LIN {X 0,Y 181.096,Z 303.588,A -85,B 0,C 180,E1 -24675.57,E2 -24675.57} C_VEL
LIN {X 0,Y 183.725,Z 307.761,A -85,B 0,C 180,E1 -24677.82,E2 -24677.82} C_VEL
LIN {X 0,Y 187.642,Z 314.233,A -85,B 0,C 180,E1 -24680.781,E2 -24680.781} C_VEL
LIN {X 0,Y 192.444,Z 323.016,A -85,B 0,C 180,E1 -24683.954,E2 -24683.954} C_VEL
LIN {X 0,Y 193.88,Z 325.932,A -85,B 0,C 180,E1 -24684.834,E2 -24684.834} C_VEL
LIN {X 0,Y 191.762,Z 350.553,A -85,B 0,C 180,E1 -24685.67,E2 -24685.67} C_VEL
LIN {X 0,Y 189.631,Z 363.427,A -85,B 0,C 180,E1 -24686.415,E2 -24686.415} C_VEL
LIN {X 0,Y 186.579,Z 375.788,A -85,B 0,C 180,E1 -24687.439,E2 -24687.439} C_VEL
LIN {X 0,Y 182.556,Z 388.05,A -85,B 0,C 180,E1 -24688.863,E2 -24688.863} C_VEL
LIN {X 0,Y 178.131,Z 398.759,A -85,B 0,C 180,E1 -24690.531,E2 -24690.531} C_VEL
LIN {X 0,Y 173.052,Z 408.926,A -85,B 0,C 180,E1 -24692.579,E2 -24692.579} C_VEL
LIN {X 0,Y 167.41,Z 418.371,A -85,B 0,C 180,E1 -24695.058,E2 -24695.058} C_VEL
LIN {X 0,Y 161.166,Z 427.427,A -85,B 0,C 180,E1 -24698.291,E2 -24698.291} C_VEL
LIN {X 0,Y 155.369,Z 434.616,A -85,B 0,C 180,E1 -24701.728,E2 -24701.728} C_VEL
LIN {X 0,Y 150.26,Z 440.26,A -85,B 0,C 180,E1 -24705.45,E2 -24705.45} C_VEL
LIN {X 0,Y 145.741,Z 444.612,A -85,B 0,C 180,E1 -24709.387,E2 -24709.387} C_VEL
LIN {X 0,Y 141.866,Z 447.811,A -85,B 0,C 180,E1 -24713.529,E2 -24713.529} C_VEL
LIN {X 0,Y 139.709,Z 449.369,A -85,B 0,C 180,E1 -24716.407,E2 -24716.407} C_VEL
LIN {X 0,Y 137.256,Z 450.755,A -85,B 0,C 180,E1 -24720.514,E2 -24720.514} C_VEL
LIN {X 0,Y 135.153,Z 451.346,A -85,B 0,C 180,E1 -24725.421,E2 -24725.421} C_VEL
LIN {X 0,Y 133.809,Z 450.698,A -85,B 0,C 180,E1 -24730.983,E2 -24730.983} C_VEL
LIN {X 0,Y 133.388,Z 449.493,A -85,B 0,C 180,E1 -24734.729,E2 -24734.729} C_VEL
LIN {X 0,Y 133.321,Z 448.048,A -85,B 0,C 180,E1 -24737.831,E2 -24737.831} C_VEL
LIN {X 0,Y 133.812,Z 445.016,A -85,B 0,C 180,E1 -24742.458,E2 -24742.458} C_VEL
LIN {X 0,Y 134.775,Z 440.923,A -85,B 0,C 180,E1 -24747.014,E2 -24747.014} C_VEL
LIN {X 0,Y 136.471,Z 434.662,A -85,B 0,C 180,E1 -24752.217,E2 -24752.217} C_VEL
LIN {X 0,Y 138.593,Z 427.846,A -85,B 0,C 180,E1 -24756.555,E2 -24756.555} C_VEL
LIN {X 0,Y 141.366,Z 419.285,A -85,B 0,C 180,E1 -24760.748,E2 -24760.748} C_VEL
LIN {X 0,Y 144.499,Z 409.445,A -85,B 0,C 180,E1 -24764.473,E2 -24764.473} C_VEL
LIN {X 0,Y 147.424,Z 399.807,A -85,B 0,C 180,E1 -24767.293,E2 -24767.293} C_VEL
LIN {X 0,Y 150.331,Z 388.712,A -85,B 0,C 180,E1 -24769.815,E2 -24769.815} C_VEL
LIN {X 0,Y 152.82,Z 376.588,A -85,B 0,C 180,E1 -24771.944,E2 -24771.944} C_VEL
LIN {X 0,Y 154.786,Z 365,A -85,B 0,C 180,E1 -24773.412,E2 -24773.412} C_VEL
LIN {X 0,Y 156.38,Z 351.822,A -85,B 0,C 180,E1 -24774.555,E2 -24774.555} C_VEL
LIN {X 0,Y 157.472,Z 336.902,A -85,B 0,C 180,E1 -24775.295,E2 -24775.295} C_VEL
LIN {X 0,Y 159.848,Z 295.992,A -85,B 0,C 180,E1 -24776.933,E2 -24776.933} C_VEL
LIN {X 0,Y 157.515,Z 290.307,A -85,B 0,C 180,E1 -24777.849,E2 -24777.849} C_VEL
LIN {X 0,Y 151.057,Z 277.224,A -85,B 0,C 180,E1 -24780.433,E2 -24780.433} C_VEL
LIN {X 0,Y 143.732,Z 264.819,A -85,B 0,C 180,E1 -24783.62,E2 -24783.62} C_VEL
LIN {X 0,Y 141.087,Z 260.921,A -85,B 0,C 180,E1 -24784.855,E2 -24784.855} C_VEL
LIN {X 0,Y 138.626,Z 257.169,A -85,B 0,C 180,E1 -24786.079,E2 -24786.079} C_VEL
LIN {X 0,Y 136.758,Z 254.919,A -85,B 0,C 180,E1 -24787.006,E2 -24787.006} C_VEL
LIN {X 0,Y 136.034,Z 252.53,A -85,B 0,C 180,E1 -24787.53,E2 -24787.53} C_VEL
LIN {X 0,Y 135.984,Z 252.525,A -85,B 0,C 180,E1 -24793.65,E2 -24793.65} C_VEL
LIN {X 0,Y 135.989,Z 252.541,A -85,B 0,C 180,E1 -24797.789,E2 -24797.789} C_VEL
LIN {X 0,Y 136.026,Z 252.509,A -85,B 0,C 180,E1 -24801.683,E2 -24801.683} C_VEL
LIN {X 0,Y 136.061,Z 252.533,A -85,B 0,C 180,E1 -24805.741,E2 -24805.741} C_VEL
LIN {X 0,Y 136.344,Z 252.463,A -85,B 0,C 180,E1 -24810.946,E2 -24810.946} C_VEL
LIN {X 0,Y 139.989,Z 268.771,A -85,B 0,C 180,E1 -24812.601,E2 -24812.601} C_VEL
LIN {X 0,Y 142.664,Z 279.155,A -85,B 0,C 180,E1 -24813.601,E2 -24813.601} C_VEL
LIN {X 0,Y 139.563,Z 347.819,A -85,B 0,C 180,E1 -24820.511,E2 -24820.511} C_VEL
LIN {X 0,Y 138.874,Z 361.236,A -85,B 0,C 180,E1 -24822.323,E2 -24822.323} C_VEL
LIN {X 0,Y 137.939,Z 375.222,A -85,B 0,C 180,E1 -24824.863,E2 -24824.863} C_VEL
LIN {X 0,Y 137.171,Z 388.146,A -85,B 0,C 180,E1 -24827.906,E2 -24827.906} C_VEL
LIN {X 0,Y 136.431,Z 400.193,A -85,B 0,C 180,E1 -24831.482,E2 -24831.482} C_VEL
LIN {X 0,Y 136.056,Z 409.375,A -85,B 0,C 180,E1 -24834.813,E2 -24834.813} C_VEL
LIN {X 0,Y 135.846,Z 419.39,A -85,B 0,C 180,E1 -24839.258,E2 -24839.258} C_VEL
LIN {X 0,Y 135.797,Z 427.45,A -85,B 0,C 180,E1 -24843.709,E2 -24843.709} C_VEL
LIN {X 0,Y 136.499,Z 435.149,A -85,B 0,C 180,E1 -24848.885,E2 -24848.885} C_VEL
LIN {X 0,Y 137.925,Z 441.004,A -85,B 0,C 180,E1 -24853.702,E2 -24853.702} C_VEL
LIN {X 0,Y 140.845,Z 446.332,A -85,B 0,C 180,E1 -24858.925,E2 -24858.925} C_VEL
LIN {X 0,Y 144.451,Z 449.823,A -85,B 0,C 180,E1 -24862.906,E2 -24862.906} C_VEL
LIN {X 0,Y 150.485,Z 453.338,A -85,B 0,C 180,E1 -24867.841,E2 -24867.841} C_VEL
LIN {X 0,Y 157.818,Z 455.582,A -85,B 0,C 180,E1 -24872.302,E2 -24872.302} C_VEL
LIN {X 0,Y 166.371,Z 456.6,A -85,B 0,C 180,E1 -24876.256,E2 -24876.256} C_VEL
LIN {X 0,Y 175.918,Z 456.39,A -85,B 0,C 180,E1 -24879.732,E2 -24879.732} C_VEL
LIN {X 0,Y 186.402,Z 454.92,A -85,B 0,C 180,E1 -24882.739,E2 -24882.739} C_VEL
LIN {X 0,Y 184.858,Z 455.476,A -85,B 0,C 180,E1 -24883.748,E2 -24883.748} C_VEL
LIN {X 0,Y 174.305,Z 457.921,A -85,B 0,C 180,E1 -24886.726,E2 -24886.726} C_VEL
LIN {X 0,Y 164.675,Z 459.211,A -85,B 0,C 180,E1 -24890.192,E2 -24890.192} C_VEL
LIN {X 0,Y 156.122,Z 459.381,A -85,B 0,C 180,E1 -24894.179,E2 -24894.179} C_VEL
LIN {X 0,Y 149.087,Z 458.493,A -85,B 0,C 180,E1 -24898.762,E2 -24898.762} C_VEL
LIN {X 0,Y 143.43,Z 456.512,A -85,B 0,C 180,E1 -24903.829,E2 -24903.829} C_VEL
LIN {X 0,Y 139.429,Z 453.415,A -85,B 0,C 180,E1 -24909.336,E2 -24909.336} C_VEL
LIN {X 0,Y 137.239,Z 448.837,A -85,B 0,C 180,E1 -24915.635,E2 -24915.635} C_VEL
LIN {X 0,Y 135.307,Z 453.281,A -85,B 0,C 180,E1 -24919.522,E2 -24919.522} C_VEL
LIN {X 0,Y 134.113,Z 457.635,A -85,B 0,C 180,E1 -24924.66,E2 -24924.66} C_VEL
LIN {X 0,Y 134.086,Z 460.72,A -85,B 0,C 180,E1 -24929.997,E2 -24929.997} C_VEL
LIN {X 0,Y 133.697,Z 462.053,A -85,B 0,C 180,E1 -24933.976,E2 -24933.976} C_VEL
LIN {X 0,Y 132.967,Z 462.531,A -85,B 0,C 180,E1 -24936.491,E2 -24936.491} C_VEL
LIN {X 0,Y 130.508,Z 462.645,A -85,B 0,C 180,E1 -24940.674,E2 -24940.674} C_VEL
LIN {X 0,Y 128.888,Z 462.263,A -85,B 0,C 180,E1 -24944.118,E2 -24944.118} C_VEL
LIN {X 0,Y 128.744,Z 461.738,A -85,B 0,C 180,E1 -24946.746,E2 -24946.746} C_VEL
LIN {X 0,Y 129.013,Z 461.468,A -85,B 0,C 180,E1 -24947.611,E2 -24947.611} C_VEL
LIN {X 0,Y 131.421,Z 459.832,A -85,B 0,C 180,E1 -24951.98,E2 -24951.98} C_VEL
LIN {X 0,Y 134.738,Z 457.195,A -85,B 0,C 180,E1 -24956.315,E2 -24956.315} C_VEL
LIN {X 0,Y 139.233,Z 453.074,A -85,B 0,C 180,E1 -24960.897,E2 -24960.897} C_VEL
LIN {X 0,Y 145.186,Z 447.039,A -85,B 0,C 180,E1 -24965.509,E2 -24965.509} C_VEL
LIN {X 0,Y 150.9,Z 440.622,A -85,B 0,C 180,E1 -24968.954,E2 -24968.954} C_VEL
LIN {X 0,Y 157.14,Z 432.662,A -85,B 0,C 180,E1 -24972.13,E2 -24972.13} C_VEL
LIN {X 0,Y 162.721,Z 424.557,A -85,B 0,C 180,E1 -24974.571,E2 -24974.571} C_VEL
LIN {X 0,Y 168.557,Z 414.679,A -85,B 0,C 180,E1 -24976.854,E2 -24976.854} C_VEL
LIN {X 0,Y 173.526,Z 404.9,A -85,B 0,C 180,E1 -24978.523,E2 -24978.523} C_VEL
LIN {X 0,Y 178.054,Z 394.302,A -85,B 0,C 180,E1 -24979.881,E2 -24979.881} C_VEL
LIN {X 0,Y 182.319,Z 381.64,A -85,B 0,C 180,E1 -24981.085,E2 -24981.085} C_VEL
LIN {X 0,Y 185.37,Z 369.086,A -85,B 0,C 180,E1 -24981.926,E2 -24981.926} C_VEL
LIN {X 0,Y 187.487,Z 355.083,A -85,B 0,C 180,E1 -24982.545,E2 -24982.545} C_VEL
LIN {X 0,Y 189.689,Z 328.895,A -85,B 0,C 180,E1 -24983.386,E2 -24983.386} C_VEL
LIN {X 0,Y 185.015,Z 319.976,A -85,B 0,C 180,E1 -24986.684,E2 -24986.684} C_VEL
LIN {X 0,Y 180.62,Z 312.326,A -85,B 0,C 180,E1 -24990.306,E2 -24990.306} C_VEL
LIN {X 0,Y 177.664,Z 307.74,A -85,B 0,C 180,E1 -24993.13,E2 -24993.13} C_VEL
LIN {X 0,Y 175.509,Z 304.331,A -85,B 0,C 180,E1 -24995.529,E2 -24995.529} C_VEL
LIN {X 0,Y 172.884,Z 300.402,A -85,B 0,C 180,E1 -24999.032,E2 -24999.032} C_VEL
LIN {X 0,Y 170.532,Z 297.011,A -85,B 0,C 180,E1 -25003.333,E2 -25003.333} C_VEL
LIN {X 0,Y 170.145,Z 295.915,A -85,B 0,C 180,E1 -25004.387,E2 -25004.387} C_VEL
LIN {X 0,Y 168.283,Z 294.151,A -85,B 0,C 180,E1 -25012.803,E2 -25012.803} C_VEL
LIN {X 0,Y 169.241,Z 294.8,A -85,B 0,C 180,E1 -25019.406,E2 -25019.406} C_VEL
LIN {X 0,Y 170.437,Z 295.952,A -85,B 0,C 180,E1 -25022.622,E2 -25022.622} C_VEL
LIN {X 0,Y 172.46,Z 299.6,A -85,B 0,C 180,E1 -25026.66,E2 -25026.66} C_VEL
LIN {X 0,Y 173.366,Z 300.816,A -85,B 0,C 180,E1 -25028.037,E2 -25028.037} C_VEL
LIN {X 0,Y 176.39,Z 305.524,A -85,B 0,C 180,E1 -25031.874,E2 -25031.874} C_VEL
LIN {X 0,Y 179.488,Z 310.456,A -85,B 0,C 180,E1 -25035.052,E2 -25035.052} C_VEL
LIN {X 0,Y 182.92,Z 316.095,A -85,B 0,C 180,E1 -25038.046,E2 -25038.046} C_VEL
LIN {X 0,Y 187.493,Z 324.427,A -85,B 0,C 180,E1 -25041.509,E2 -25041.509} C_VEL
LIN {X 0,Y 189.89,Z 329.186,A -85,B 0,C 180,E1 -25043.138,E2 -25043.138} C_VEL
LIN {X 0,Y 187.851,Z 351.434,A -85,B 0,C 180,E1 -25043.902,E2 -25043.902} C_VEL
LIN {X 0,Y 185.479,Z 364.794,A -85,B 0,C 180,E1 -25044.682,E2 -25044.682} C_VEL
LIN {X 0,Y 182.301,Z 377.03,A -85,B 0,C 180,E1 -25045.719,E2 -25045.719} C_VEL
LIN {X 0,Y 178.461,Z 388.166,A -85,B 0,C 180,E1 -25047.007,E2 -25047.007} C_VEL
LIN {X 0,Y 173.315,Z 400.117,A -85,B 0,C 180,E1 -25048.888,E2 -25048.888} C_VEL
LIN {X 0,Y 167.981,Z 410.175,A -85,B 0,C 180,E1 -25050.948,E2 -25050.948} C_VEL
LIN {X 0,Y 162.142,Z 419.412,A -85,B 0,C 180,E1 -25053.453,E2 -25053.453} C_VEL
LIN {X 0,Y 156.702,Z 426.977,A -85,B 0,C 180,E1 -25056.173,E2 -25056.173} C_VEL
LIN {X 0,Y 150.543,Z 434.333,A -85,B 0,C 180,E1 -25059.625,E2 -25059.625} C_VEL
LIN {X 0,Y 145.051,Z 440.122,A -85,B 0,C 180,E1 -25063.388,E2 -25063.388} C_VEL
LIN {X 0,Y 140.179,Z 444.582,A -85,B 0,C 180,E1 -25067.408,E2 -25067.408} C_VEL
LIN {X 0,Y 135.963,Z 447.881,A -85,B 0,C 180,E1 -25071.667,E2 -25071.667} C_VEL
LIN {X 0,Y 133.589,Z 449.487,A -85,B 0,C 180,E1 -25074.645,E2 -25074.645} C_VEL
LIN {X 0,Y 130.542,Z 451.105,A -85,B 0,C 180,E1 -25079.476,E2 -25079.476} C_VEL
LIN {X 0,Y 128.462,Z 451.649,A -85,B 0,C 180,E1 -25084.049,E2 -25084.049} C_VEL
LIN {X 0,Y 127.463,Z 451.532,A -85,B 0,C 180,E1 -25087.3,E2 -25087.3} C_VEL
LIN {X 0,Y 126.782,Z 450.959,A -85,B 0,C 180,E1 -25090.577,E2 -25090.577} C_VEL
LIN {X 0,Y 126.351,Z 449.974,A -85,B 0,C 180,E1 -25093.856,E2 -25093.856} C_VEL
LIN {X 0,Y 126.205,Z 448.588,A -85,B 0,C 180,E1 -25097.133,E2 -25097.133} C_VEL
LIN {X 0,Y 126.637,Z 445.649,A -85,B 0,C 180,E1 -25102.028,E2 -25102.028} C_VEL
LIN {X 0,Y 127.621,Z 441.664,A -85,B 0,C 180,E1 -25106.847,E2 -25106.847} C_VEL
LIN {X 0,Y 129.342,Z 435.529,A -85,B 0,C 180,E1 -25112.339,E2 -25112.339} C_VEL
LIN {X 0,Y 131.504,Z 428.835,A -85,B 0,C 180,E1 -25116.91,E2 -25116.91} C_VEL
LIN {X 0,Y 134.369,Z 420.486,A -85,B 0,C 180,E1 -25121.315,E2 -25121.315} C_VEL
LIN {X 0,Y 137.27,Z 411.874,A -85,B 0,C 180,E1 -25124.836,E2 -25124.836} C_VEL
LIN {X 0,Y 140.634,Z 401.515,A -85,B 0,C 180,E1 -25128.126,E2 -25128.126} C_VEL
LIN {X 0,Y 143.692,Z 390.708,A -85,B 0,C 180,E1 -25130.772,E2 -25130.772} C_VEL
LIN {X 0,Y 146.362,Z 378.969,A -85,B 0,C 180,E1 -25132.967,E2 -25132.967} C_VEL
LIN {X 0,Y 148.242,Z 368.163,A -85,B 0,C 180,E1 -25134.512,E2 -25134.512} C_VEL
LIN {X 0,Y 150.067,Z 355.774,A -85,B 0,C 180,E1 -25135.732,E2 -25135.732} C_VEL
LIN {X 0,Y 151.278,Z 342.381,A -85,B 0,C 180,E1 -25136.538,E2 -25136.538} C_VEL
LIN {X 0,Y 153.907,Z 297.378,A -85,B 0,C 180,E1 -25138.42,E2 -25138.42} C_VEL
LIN {X 0,Y 146.974,Z 282.62,A -85,B 0,C 180,E1 -25141.373,E2 -25141.373} C_VEL
LIN {X 0,Y 139.613,Z 269.819,A -85,B 0,C 180,E1 -25144.797,E2 -25144.797} C_VEL
LIN {X 0,Y 134.581,Z 262.349,A -85,B 0,C 180,E1 -25147.376,E2 -25147.376} C_VEL
LIN {X 0,Y 132.346,Z 258.968,A -85,B 0,C 180,E1 -25148.626,E2 -25148.626} C_VEL
LIN {X 0,Y 129.679,Z 255.773,A -85,B 0,C 180,E1 -25150.144,E2 -25150.144} C_VEL
LIN {X 0,Y 128.928,Z 253.414,A -85,B 0,C 180,E1 -25150.751,E2 -25150.751} C_VEL
LIN {X 0,Y 128.918,Z 253.415,A -85,B 0,C 180,E1 -25155.134,E2 -25155.134} C_VEL
LIN {X 0,Y 128.94,Z 253.397,A -85,B 0,C 180,E1 -25159.742,E2 -25159.742} C_VEL
LIN {X 0,Y 128.964,Z 253.412,A -85,B 0,C 180,E1 -25164.835,E2 -25164.835} C_VEL
LIN {X 0,Y 129.318,Z 253.337,A -85,B 0,C 180,E1 -25170.947,E2 -25170.947} C_VEL
LIN {X 0,Y 132.682,Z 268.752,A -85,B 0,C 180,E1 -25172.595,E2 -25172.595} C_VEL
LIN {X 0,Y 135.523,Z 279.836,A -85,B 0,C 180,E1 -25173.708,E2 -25173.708} C_VEL
LIN {X 0,Y 132.528,Z 349.023,A -85,B 0,C 180,E1 -25181.145,E2 -25181.145} C_VEL
LIN {X 0,Y 131.76,Z 362.486,A -85,B 0,C 180,E1 -25183.141,E2 -25183.141} C_VEL
LIN {X 0,Y 131,Z 374.658,A -85,B 0,C 180,E1 -25185.5,E2 -25185.5} C_VEL
LIN {X 0,Y 130.285,Z 387.768,A -85,B 0,C 180,E1 -25188.723,E2 -25188.723} C_VEL
LIN {X 0,Y 129.592,Z 400.118,A -85,B 0,C 180,E1 -25192.599,E2 -25192.599} C_VEL
LIN {X 0,Y 129.317,Z 409.284,A -85,B 0,C 180,E1 -25196.104,E2 -25196.104} C_VEL
LIN {X 0,Y 129.172,Z 419.182,A -85,B 0,C 180,E1 -25200.779,E2 -25200.779} C_VEL
LIN {X 0,Y 129.231,Z 427.182,A -85,B 0,C 180,E1 -25205.46,E2 -25205.46} C_VEL
LIN {X 0,Y 130,Z 433.861,A -85,B 0,C 180,E1 -25210.119,E2 -25210.119} C_VEL
LIN {X 0,Y 131.719,Z 440.251,A -85,B 0,C 180,E1 -25215.472,E2 -25215.472} C_VEL
LIN {X 0,Y 134.293,Z 444.828,A -85,B 0,C 180,E1 -25219.886,E2 -25219.886} C_VEL
LIN {X 0,Y 139.442,Z 449.767,A -85,B 0,C 180,E1 -25225.366,E2 -25225.366} C_VEL
LIN {X 0,Y 144.281,Z 452.64,A -85,B 0,C 180,E1 -25229.15,E2 -25229.15} C_VEL
LIN {X 0,Y 151.88,Z 455.357,A -85,B 0,C 180,E1 -25233.73,E2 -25233.73} C_VEL
LIN {X 0,Y 160.706,Z 456.885,A -85,B 0,C 180,E1 -25237.752,E2 -25237.752} C_VEL
LIN {X 0,Y 170.536,Z 457.214,A -85,B 0,C 180,E1 -25241.252,E2 -25241.252} C_VEL
LIN {X 0,Y 175.825,Z 456.918,A -85,B 0,C 180,E1 -25242.805,E2 -25242.805} C_VEL
LIN {X 0,Y 174.519,Z 457.227,A -85,B 0,C 180,E1 -25243.539,E2 -25243.539} C_VEL
LIN {X 0,Y 164.125,Z 458.559,A -85,B 0,C 180,E1 -25246.75,E2 -25246.75} C_VEL
LIN {X 0,Y 154.73,Z 458.793,A -85,B 0,C 180,E1 -25250.51,E2 -25250.51} C_VEL
LIN {X 0,Y 146.633,Z 457.986,A -85,B 0,C 180,E1 -25254.886,E2 -25254.886} C_VEL
LIN {X 0,Y 140.03,Z 456.151,A -85,B 0,C 180,E1 -25259.871,E2 -25259.871} C_VEL
LIN {X 0,Y 134.92,Z 453.212,A -85,B 0,C 180,E1 -25265.369,E2 -25265.369} C_VEL
LIN {X 0,Y 131.765,Z 449.188,A -85,B 0,C 180,E1 -25271.332,E2 -25271.332} C_VEL
LIN {X 0,Y 131.002,Z 447.063,A -85,B 0,C 180,E1 -25274.038,E2 -25274.038} C_VEL
LIN {X 0,Y 128.347,Z 452.655,A -85,B 0,C 180,E1 -25278.947,E2 -25278.947} C_VEL
LIN {X 0,Y 127.011,Z 457.438,A -85,B 0,C 180,E1 -25284.877,E2 -25284.877} C_VEL
LIN {X 0,Y 126.994,Z 460.252,A -85,B 0,C 180,E1 -25289.997,E2 -25289.997} C_VEL
LIN {X 0,Y 126.631,Z 461.567,A -85,B 0,C 180,E1 -25293.888,E2 -25293.888} C_VEL
LIN {X 0,Y 126.832,Z 462.445,A -85,B 0,C 180,E1 -25299.565,E2 -25299.565} C_VEL
LIN {X 0,Y 128.346,Z 461.938,A -85,B 0,C 180,E1 -25305.886,E2 -25305.886} C_VEL
LIN {X 0,Y 129.013,Z 461.468,A -85,B 0,C 180,E1 -25307.611,E2 -25307.611} C_VEL
LIN {X 0,Y 129.609,Z 460.66,A -85,B 0,C 180,E1 -25310.193,E2 -25310.193} C_VEL
LIN {X 0,Y 129.498,Z 458.803,A -85,B 0,C 180,E1 -25314.502,E2 -25314.502} C_VEL
LIN {X 0,Y 129.785,Z 456.84,A -85,B 0,C 180,E1 -25317.902,E2 -25317.902} C_VEL
LIN {X 0,Y 130.986,Z 455.063,A -85,B 0,C 180,E1 -25320.324,E2 -25320.324} C_VEL
LIN {X 0,Y 131.666,Z 454.396,A -85,B 0,C 180,E1 -25321.079,E2 -25321.079} C_VEL
LIN {X 0,Y 137.627,Z 448.923,A -85,B 0,C 180,E1 -25325.958,E2 -25325.958} C_VEL
LIN {X 0,Y 144.416,Z 441.951,A -85,B 0,C 180,E1 -25330.147,E2 -25330.147} C_VEL
LIN {X 0,Y 150.835,Z 434.432,A -85,B 0,C 180,E1 -25333.409,E2 -25333.409} C_VEL
LIN {X 0,Y 157.764,Z 424.998,A -85,B 0,C 180,E1 -25336.373,E2 -25336.373} C_VEL
LIN {X 0,Y 163.796,Z 415.291,A -85,B 0,C 180,E1 -25338.662,E2 -25338.662} C_VEL
LIN {X 0,Y 168.932,Z 405.76,A -85,B 0,C 180,E1 -25340.318,E2 -25340.318} C_VEL
LIN {X 0,Y 173.584,Z 395.478,A -85,B 0,C 180,E1 -25341.665,E2 -25341.665} C_VEL
LIN {X 0,Y 178.035,Z 383.038,A -85,B 0,C 180,E1 -25342.864,E2 -25342.864} C_VEL
LIN {X 0,Y 181.47,Z 370.014,A -85,B 0,C 180,E1 -25343.762,E2 -25343.762} C_VEL
LIN {X 0,Y 183.628,Z 357.081,A -85,B 0,C 180,E1 -25344.358,E2 -25344.358} C_VEL
LIN {X 0,Y 185.849,Z 332.311,A -85,B 0,C 180,E1 -25345.175,E2 -25345.175} C_VEL
LIN {X 0,Y 181.843,Z 324.399,A -85,B 0,C 180,E1 -25348.303,E2 -25348.303} C_VEL
LIN {X 0,Y 177.856,Z 317.389,A -85,B 0,C 180,E1 -25351.899,E2 -25351.899} C_VEL
LIN {X 0,Y 175.589,Z 313.671,A -85,B 0,C 180,E1 -25354.275,E2 -25354.275} C_VEL
LIN {X 0,Y 173.88,Z 310.837,A -85,B 0,C 180,E1 -25356.321,E2 -25356.321} C_VEL
LIN {X 0,Y 171.587,Z 307.194,A -85,B 0,C 180,E1 -25359.594,E2 -25359.594} C_VEL
LIN {X 0,Y 169.272,Z 303.528,A -85,B 0,C 180,E1 -25364.202,E2 -25364.202} C_VEL
LIN {X 0,Y 168.936,Z 302.786,A -85,B 0,C 180,E1 -25365.154,E2 -25365.154} C_VEL
LIN {X 0,Y 167.406,Z 301.202,A -85,B 0,C 180,E1 -25372.765,E2 -25372.765} C_VEL
LIN {X 0,Y 168.187,Z 301.698,A -85,B 0,C 180,E1 -25378.803,E2 -25378.803} C_VEL
LIN {X 0,Y 169.358,Z 302.973,A -85,B 0,C 180,E1 -25382.23,E2 -25382.23} C_VEL
LIN {X 0,Y 171.337,Z 306.563,A -85,B 0,C 180,E1 -25386.339,E2 -25386.339} C_VEL
LIN {X 0,Y 172.146,Z 307.838,A -85,B 0,C 180,E1 -25387.643,E2 -25387.643} C_VEL
LIN {X 0,Y 174.846,Z 312.263,A -85,B 0,C 180,E1 -25391.25,E2 -25391.25} C_VEL
LIN {X 0,Y 177.716,Z 316.998,A -85,B 0,C 180,E1 -25394.345,E2 -25394.345} C_VEL
LIN {X 0,Y 180.999,Z 322.739,A -85,B 0,C 180,E1 -25397.368,E2 -25397.368} C_VEL
LIN {X 0,Y 184.887,Z 330.157,A -85,B 0,C 180,E1 -25400.485,E2 -25400.485} C_VEL
LIN {X 0,Y 186.044,Z 332.539,A -85,B 0,C 180,E1 -25401.344,E2 -25401.344} C_VEL
LIN {X 0,Y 184.115,Z 352.442,A -85,B 0,C 180,E1 -25402.064,E2 -25402.064} C_VEL
LIN {X 0,Y 181.69,Z 365.44,A -85,B 0,C 180,E1 -25402.824,E2 -25402.824} C_VEL
LIN {X 0,Y 178.376,Z 377.673,A -85,B 0,C 180,E1 -25403.859,E2 -25403.859} C_VEL
LIN {X 0,Y 174.567,Z 388.29,A -85,B 0,C 180,E1 -25405.07,E2 -25405.07} C_VEL
LIN {X 0,Y 169.5,Z 399.721,A -85,B 0,C 180,E1 -25406.838,E2 -25406.838} C_VEL
LIN {X 0,Y 163.682,Z 410.366,A -85,B 0,C 180,E1 -25408.98,E2 -25408.98} C_VEL
LIN {X 0,Y 158.194,Z 418.806,A -85,B 0,C 180,E1 -25411.223,E2 -25411.223} C_VEL
LIN {X 0,Y 152.422,Z 426.523,A -85,B 0,C 180,E1 -25413.911,E2 -25413.911} C_VEL
LIN {X 0,Y 145.943,Z 434.018,A -85,B 0,C 180,E1 -25417.391,E2 -25417.391} C_VEL
LIN {X 0,Y 140.062,Z 439.965,A -85,B 0,C 180,E1 -25421.183,E2 -25421.183} C_VEL
LIN {X 0,Y 134.806,Z 444.551,A -85,B 0,C 180,E1 -25425.271,E2 -25425.271} C_VEL
LIN {X 0,Y 130.219,Z 447.951,A -85,B 0,C 180,E1 -25429.64,E2 -25429.64} C_VEL
LIN {X 0,Y 127.592,Z 449.605,A -85,B 0,C 180,E1 -25432.711,E2 -25432.711} C_VEL
LIN {X 0,Y 123.885,Z 451.452,A -85,B 0,C 180,E1 -25438.317,E2 -25438.317} C_VEL
LIN {X 0,Y 121.86,Z 451.951,A -85,B 0,C 180,E1 -25442.528,E2 -25442.528} C_VEL
LIN {X 0,Y 120.686,Z 451.881,A -85,B 0,C 180,E1 -25445.948,E2 -25445.948} C_VEL
LIN {X 0,Y 119.768,Z 451.284,A -85,B 0,C 180,E1 -25449.869,E2 -25449.869} C_VEL
LIN {X 0,Y 119.106,Z 449.114,A -85,B 0,C 180,E1 -25456.352,E2 -25456.352} C_VEL
LIN {X 0,Y 119.445,Z 446.268,A -85,B 0,C 180,E1 -25461.545,E2 -25461.545} C_VEL
LIN {X 0,Y 120.433,Z 442.377,A -85,B 0,C 180,E1 -25466.658,E2 -25466.658} C_VEL
LIN {X 0,Y 121.895,Z 437.363,A -85,B 0,C 180,E1 -25471.656,E2 -25471.656} C_VEL
LIN {X 0,Y 123.96,Z 431.05,A -85,B 0,C 180,E1 -25476.514,E2 -25476.514} C_VEL
LIN {X 0,Y 126.835,Z 423.124,A -85,B 0,C 180,E1 -25481.186,E2 -25481.186} C_VEL
LIN {X 0,Y 129.789,Z 415.03,A -85,B 0,C 180,E1 -25484.908,E2 -25484.908} C_VEL
LIN {X 0,Y 133.171,Z 405.167,A -85,B 0,C 180,E1 -25488.464,E2 -25488.464} C_VEL
LIN {X 0,Y 136.615,Z 394.013,A -85,B 0,C 180,E1 -25491.506,E2 -25491.506} C_VEL
LIN {X 0,Y 139.476,Z 383.129,A -85,B 0,C 180,E1 -25493.776,E2 -25493.776} C_VEL
LIN {X 0,Y 141.798,Z 371.195,A -85,B 0,C 180,E1 -25495.705,E2 -25495.705} C_VEL
LIN {X 0,Y 143.998,Z 357.851,A -85,B 0,C 180,E1 -25497.127,E2 -25497.127} C_VEL
LIN {X 0,Y 145.335,Z 344.548,A -85,B 0,C 180,E1 -25498.034,E2 -25498.034} C_VEL
LIN {X 0,Y 148.122,Z 299.482,A -85,B 0,C 180,E1 -25499.968,E2 -25499.968} C_VEL
LIN {X 0,Y 141.994,Z 286.3,A -85,B 0,C 180,E1 -25502.804,E2 -25502.804} C_VEL
LIN {X 0,Y 135.309,Z 274.467,A -85,B 0,C 180,E1 -25506.171,E2 -25506.171} C_VEL
LIN {X 0,Y 130.66,Z 267.479,A -85,B 0,C 180,E1 -25508.731,E2 -25508.731} C_VEL
LIN {X 0,Y 127.837,Z 263.403,A -85,B 0,C 180,E1 -25510.423,E2 -25510.423} C_VEL
LIN {X 0,Y 125.684,Z 260.37,A -85,B 0,C 180,E1 -25511.799,E2 -25511.799} C_VEL
LIN {X 0,Y 125.114,Z 259.446,A -85,B 0,C 180,E1 -25512.189,E2 -25512.189} C_VEL
LIN {X 0,Y 122.903,Z 257.284,A -85,B 0,C 180,E1 -25513.631,E2 -25513.631} C_VEL
LIN {X 0,Y 121.961,Z 254.883,A -85,B 0,C 180,E1 -25514.417,E2 -25514.417} C_VEL
LIN {X 0,Y 121.862,Z 254.288,A -85,B 0,C 180,E1 -25514.635,E2 -25514.635} C_VEL
LIN {X 0,Y 121.858,Z 254.273,A -85,B 0,C 180,E1 -25520.623,E2 -25520.623} C_VEL
LIN {X 0,Y 121.915,Z 254.288,A -85,B 0,C 180,E1 -25524.796,E2 -25524.796} C_VEL
LIN {X 0,Y 122.3,Z 254.373,A -85,B 0,C 180,E1 -25531.059,E2 -25531.059} C_VEL
LIN {X 0,Y 125.697,Z 269.93,A -85,B 0,C 180,E1 -25532.763,E2 -25532.763} C_VEL
LIN {X 0,Y 128.368,Z 280.717,A -85,B 0,C 180,E1 -25533.906,E2 -25533.906} C_VEL
LIN {X 0,Y 125.574,Z 348.831,A -85,B 0,C 180,E1 -25541.735,E2 -25541.735} C_VEL
LIN {X 0,Y 124.813,Z 362.935,A -85,B 0,C 180,E1 -25543.942,E2 -25543.942} C_VEL
LIN {X 0,Y 123.99,Z 375.679,A -85,B 0,C 180,E1 -25546.617,E2 -25546.617} C_VEL
LIN {X 0,Y 123.424,Z 387.576,A -85,B 0,C 180,E1 -25549.749,E2 -25549.749} C_VEL
LIN {X 0,Y 122.87,Z 398.752,A -85,B 0,C 180,E1 -25553.43,E2 -25553.43} C_VEL
LIN {X 0,Y 122.612,Z 408.977,A -85,B 0,C 180,E1 -25557.535,E2 -25557.535} C_VEL
LIN {X 0,Y 122.569,Z 417.358,A -85,B 0,C 180,E1 -25561.642,E2 -25561.642} C_VEL
LIN {X 0,Y 122.701,Z 425.598,A -85,B 0,C 180,E1 -25566.577,E2 -25566.577} C_VEL
LIN {X 0,Y 123.831,Z 433.495,A -85,B 0,C 180,E1 -25572.288,E2 -25572.288} C_VEL
LIN {X 0,Y 125.923,Z 439.912,A -85,B 0,C 180,E1 -25577.876,E2 -25577.876} C_VEL
LIN {X 0,Y 130.349,Z 445.98,A -85,B 0,C 180,E1 -25583.851,E2 -25583.851} C_VEL
LIN {X 0,Y 136.418,Z 450.724,A -85,B 0,C 180,E1 -25589.302,E2 -25589.302} C_VEL
LIN {X 0,Y 141.932,Z 453.456,A -85,B 0,C 180,E1 -25593.002,E2 -25593.002} C_VEL
LIN {X 0,Y 150.411,Z 456.07,A -85,B 0,C 180,E1 -25597.403,E2 -25597.403} C_VEL
LIN {X 0,Y 160.081,Z 457.521,A -85,B 0,C 180,E1 -25601.188,E2 -25601.188} C_VEL
LIN {X 0,Y 165.268,Z 457.805,A -85,B 0,C 180,E1 -25602.874,E2 -25602.874} C_VEL
LIN {X 0,Y 164.266,Z 457.917,A -85,B 0,C 180,E1 -25603.333,E2 -25603.333} C_VEL
LIN {X 0,Y 154.093,Z 458.197,A -85,B 0,C 180,E1 -25606.829,E2 -25606.829} C_VEL
LIN {X 0,Y 144.974,Z 457.436,A -85,B 0,C 180,E1 -25610.931,E2 -25610.931} C_VEL
LIN {X 0,Y 137.36,Z 455.712,A -85,B 0,C 180,E1 -25615.746,E2 -25615.746} C_VEL
LIN {X 0,Y 131.235,Z 452.942,A -85,B 0,C 180,E1 -25621.182,E2 -25621.182} C_VEL
LIN {X 0,Y 126.859,Z 449.077,A -85,B 0,C 180,E1 -25627.179,E2 -25627.179} C_VEL
LIN {X 0,Y 124.783,Z 445.341,A -85,B 0,C 180,E1 -25632.375,E2 -25632.375} C_VEL
LIN {X 0,Y 122.102,Z 450.416,A -85,B 0,C 180,E1 -25636.685,E2 -25636.685} C_VEL
LIN {X 0,Y 120.451,Z 454.82,A -85,B 0,C 180,E1 -25641.609,E2 -25641.609} C_VEL
LIN {X 0,Y 119.791,Z 458.142,A -85,B 0,C 180,E1 -25646.633,E2 -25646.633} C_VEL
LIN {X 0,Y 119.906,Z 459.785,A -85,B 0,C 180,E1 -25649.996,E2 -25649.996} C_VEL
LIN {X 0,Y 119.597,Z 460.972,A -85,B 0,C 180,E1 -25653.365,E2 -25653.365} C_VEL
LIN {X 0,Y 119.504,Z 461.756,A -85,B 0,C 180,E1 -25656.751,E2 -25656.751} C_VEL
LIN {X 0,Y 120.477,Z 462.082,A -85,B 0,C 180,E1 -25663.49,E2 -25663.49} C_VEL
LIN {X 0,Y 122.916,Z 460.886,A -85,B 0,C 180,E1 -25670.06,E2 -25670.06} C_VEL
LIN {X 0,Y 127.097,Z 458.053,A -85,B 0,C 180,E1 -25676.251,E2 -25676.251} C_VEL
LIN {X 0,Y 131.666,Z 454.396,A -85,B 0,C 180,E1 -25681.079,E2 -25681.079} C_VEL
LIN {X 0,Y 133.453,Z 452.323,A -85,B 0,C 180,E1 -25683.341,E2 -25683.341} C_VEL
LIN {X 0,Y 135.266,Z 448.494,A -85,B 0,C 180,E1 -25687.165,E2 -25687.165} C_VEL
LIN {X 0,Y 137.595,Z 444.129,A -85,B 0,C 180,E1 -25690.749,E2 -25690.749} C_VEL
LIN {X 0,Y 140.09,Z 441.072,A -85,B 0,C 180,E1 -25692.564,E2 -25692.564} C_VEL
LIN {X 0,Y 146.936,Z 433.295,A -85,B 0,C 180,E1 -25695.84,E2 -25695.84} C_VEL
LIN {X 0,Y 154.246,Z 423.694,A -85,B 0,C 180,E1 -25698.742,E2 -25698.742} C_VEL
LIN {X 0,Y 160.557,Z 413.765,A -85,B 0,C 180,E1 -25700.978,E2 -25700.978} C_VEL
LIN {X 0,Y 165.887,Z 403.936,A -85,B 0,C 180,E1 -25702.591,E2 -25702.591} C_VEL
LIN {X 0,Y 170.712,Z 393.276,A -85,B 0,C 180,E1 -25703.89,E2 -25703.89} C_VEL
LIN {X 0,Y 175.095,Z 380.926,A -85,B 0,C 180,E1 -25705.017,E2 -25705.017} C_VEL
LIN {X 0,Y 178.374,Z 368.151,A -85,B 0,C 180,E1 -25705.828,E2 -25705.828} C_VEL
LIN {X 0,Y 180.522,Z 354.655,A -85,B 0,C 180,E1 -25706.417,E2 -25706.417} C_VEL
LIN {X 0,Y 182.272,Z 335.881,A -85,B 0,C 180,E1 -25707.002,E2 -25707.002} C_VEL
LIN {X 0,Y 178.364,Z 328.023,A -85,B 0,C 180,E1 -25710.396,E2 -25710.396} C_VEL
LIN {X 0,Y 174.718,Z 321.381,A -85,B 0,C 180,E1 -25714.137,E2 -25714.137} C_VEL
LIN {X 0,Y 172.179,Z 317.18,A -85,B 0,C 180,E1 -25717.27,E2 -25717.27} C_VEL
LIN {X 0,Y 170.348,Z 314.022,A -85,B 0,C 180,E1 -25720.101,E2 -25720.101} C_VEL
LIN {X 0,Y 168.172,Z 310.434,A -85,B 0,C 180,E1 -25724.694,E2 -25724.694} C_VEL
LIN {X 0,Y 167.929,Z 309.774,A -85,B 0,C 180,E1 -25725.458,E2 -25725.458} C_VEL
LIN {X 0,Y 166.528,Z 308.253,A -85,B 0,C 180,E1 -25732.727,E2 -25732.727} C_VEL
LIN {X 0,Y 167.38,Z 308.862,A -85,B 0,C 180,E1 -25739.098,E2 -25739.098} C_VEL
LIN {X 0,Y 168.221,Z 309.8,A -85,B 0,C 180,E1 -25741.632,E2 -25741.632} C_VEL
LIN {X 0,Y 170.686,Z 314.362,A -85,B 0,C 180,E1 -25746.821,E2 -25746.821} C_VEL
LIN {X 0,Y 173.36,Z 319.013,A -85,B 0,C 180,E1 -25750.652,E2 -25750.652} C_VEL
LIN {X 0,Y 176.52,Z 324.391,A -85,B 0,C 180,E1 -25754.177,E2 -25754.177} C_VEL
LIN {X 0,Y 180.456,Z 331.966,A -85,B 0,C 180,E1 -25757.861,E2 -25757.861} C_VEL
LIN {X 0,Y 182.427,Z 336.065,A -85,B 0,C 180,E1 -25759.501,E2 -25759.501} C_VEL
LIN {X 0,Y 180.766,Z 352.381,A -85,B 0,C 180,E1 -25760.095,E2 -25760.095} C_VEL
LIN {X 0,Y 178.225,Z 365.655,A -85,B 0,C 180,E1 -25760.855,E2 -25760.855} C_VEL
LIN {X 0,Y 174.821,Z 377.796,A -85,B 0,C 180,E1 -25761.848,E2 -25761.848} C_VEL
LIN {X 0,Y 170.889,Z 388.494,A -85,B 0,C 180,E1 -25763.052,E2 -25763.052} C_VEL
LIN {X 0,Y 165.442,Z 400.289,A -85,B 0,C 180,E1 -25764.849,E2 -25764.849} C_VEL
LIN {X 0,Y 159.595,Z 410.593,A -85,B 0,C 180,E1 -25766.914,E2 -25766.914} C_VEL
LIN {X 0,Y 153.243,Z 419.865,A -85,B 0,C 180,E1 -25769.388,E2 -25769.388} C_VEL
LIN {X 0,Y 147.245,Z 427.45,A -85,B 0,C 180,E1 -25772.097,E2 -25772.097} C_VEL
LIN {X 0,Y 140.476,Z 434.833,A -85,B 0,C 180,E1 -25775.617,E2 -25775.617} C_VEL
LIN {X 0,Y 135.277,Z 439.77,A -85,B 0,C 180,E1 -25778.81,E2 -25778.81} C_VEL
LIN {X 0,Y 129.637,Z 444.488,A -85,B 0,C 180,E1 -25782.962,E2 -25782.962} C_VEL
LIN {X 0,Y 124.665,Z 448.005,A -85,B 0,C 180,E1 -25787.434,E2 -25787.434} C_VEL
LIN {X 0,Y 121.759,Z 449.724,A -85,B 0,C 180,E1 -25790.59,E2 -25790.59} C_VEL
LIN {X 0,Y 117.266,Z 451.803,A -85,B 0,C 180,E1 -25797.042,E2 -25797.042} C_VEL
LIN {X 0,Y 115.355,Z 452.254,A -85,B 0,C 180,E1 -25800.835,E2 -25800.835} C_VEL
LIN {X 0,Y 113.983,Z 452.229,A -85,B 0,C 180,E1 -25804.435,E2 -25804.435} C_VEL
LIN {X 0,Y 112.801,Z 451.587,A -85,B 0,C 180,E1 -25809.161,E2 -25809.161} C_VEL
LIN {X 0,Y 112.027,Z 449.64,A -85,B 0,C 180,E1 -25815.471,E2 -25815.471} C_VEL
LIN {X 0,Y 112.279,Z 446.885,A -85,B 0,C 180,E1 -25821.001,E2 -25821.001} C_VEL
LIN {X 0,Y 113.246,Z 443.09,A -85,B 0,C 180,E1 -25826.446,E2 -25826.446} C_VEL
LIN {X 0,Y 114.733,Z 438.178,A -85,B 0,C 180,E1 -25831.759,E2 -25831.759} C_VEL
LIN {X 0,Y 116.863,Z 432.003,A -85,B 0,C 180,E1 -25836.912,E2 -25836.912} C_VEL
LIN {X 0,Y 119.832,Z 424.251,A -85,B 0,C 180,E1 -25841.849,E2 -25841.849} C_VEL
LIN {X 0,Y 122.919,Z 416.313,A -85,B 0,C 180,E1 -25845.762,E2 -25845.762} C_VEL
LIN {X 0,Y 126.407,Z 406.658,A -85,B 0,C 180,E1 -25849.49,E2 -25849.49} C_VEL
LIN {X 0,Y 130.037,Z 395.852,A -85,B 0,C 180,E1 -25852.652,E2 -25852.652} C_VEL
LIN {X 0,Y 133.015,Z 385.322,A -85,B 0,C 180,E1 -25855.008,E2 -25855.008} C_VEL
LIN {X 0,Y 135.665,Z 372.857,A -85,B 0,C 180,E1 -25857.167,E2 -25857.167} C_VEL
LIN {X 0,Y 137.923,Z 360.412,A -85,B 0,C 180,E1 -25858.609,E2 -25858.609} C_VEL
LIN {X 0,Y 139.418,Z 347.358,A -85,B 0,C 180,E1 -25859.603,E2 -25859.603} C_VEL
LIN {X 0,Y 142.463,Z 301.582,A -85,B 0,C 180,E1 -25861.638,E2 -25861.638} C_VEL
LIN {X 0,Y 136.464,Z 288.691,A -85,B 0,C 180,E1 -25864.679,E2 -25864.679} C_VEL
LIN {X 0,Y 130.603,Z 278.315,A -85,B 0,C 180,E1 -25867.903,E2 -25867.903} C_VEL
LIN {X 0,Y 126.403,Z 271.974,A -85,B 0,C 180,E1 -25870.424,E2 -25870.424} C_VEL
LIN {X 0,Y 124.182,Z 268.752,A -85,B 0,C 180,E1 -25871.866,E2 -25871.866} C_VEL
LIN {X 0,Y 121.726,Z 265.203,A -85,B 0,C 180,E1 -25873.575,E2 -25873.575} C_VEL
LIN {X 0,Y 119.333,Z 262.276,A -85,B 0,C 180,E1 -25875.321,E2 -25875.321} C_VEL
LIN {X 0,Y 118.453,Z 260.54,A -85,B 0,C 180,E1 -25876.067,E2 -25876.067} C_VEL
LIN {X 0,Y 116.067,Z 258.423,A -85,B 0,C 180,E1 -25877.938,E2 -25877.938} C_VEL
LIN {X 0,Y 114.947,Z 255.876,A -85,B 0,C 180,E1 -25879.052,E2 -25879.052} C_VEL
LIN {X 0,Y 114.803,Z 255.159,A -85,B 0,C 180,E1 -25879.279,E2 -25879.279} C_VEL
LIN {X 0,Y 114.869,Z 255.174,A -85,B 0,C 180,E1 -25886.588,E2 -25886.588} C_VEL
LIN {X 0,Y 115.28,Z 255.277,A -85,B 0,C 180,E1 -25891.179,E2 -25891.179} C_VEL
LIN {X 0,Y 118.673,Z 271.007,A -85,B 0,C 180,E1 -25893.007,E2 -25893.007} C_VEL
LIN {X 0,Y 121.255,Z 281.402,A -85,B 0,C 180,E1 -25894.156,E2 -25894.156} C_VEL
LIN {X 0,Y 118.637,Z 347.804,A -85,B 0,C 180,E1 -25902.325,E2 -25902.325} C_VEL
LIN {X 0,Y 117.965,Z 361.27,A -85,B 0,C 180,E1 -25904.497,E2 -25904.497} C_VEL
LIN {X 0,Y 117.273,Z 373.033,A -85,B 0,C 180,E1 -25907.012,E2 -25907.012} C_VEL
LIN {X 0,Y 116.717,Z 385.83,A -85,B 0,C 180,E1 -25910.468,E2 -25910.468} C_VEL
LIN {X 0,Y 116.202,Z 397.272,A -85,B 0,C 180,E1 -25914.359,E2 -25914.359} C_VEL
LIN {X 0,Y 116.07,Z 406.685,A -85,B 0,C 180,E1 -25918.264,E2 -25918.264} C_VEL
LIN {X 0,Y 116.058,Z 415.339,A -85,B 0,C 180,E1 -25922.602,E2 -25922.602} C_VEL
LIN {X 0,Y 116.299,Z 423.81,A -85,B 0,C 180,E1 -25927.814,E2 -25927.814} C_VEL
LIN {X 0,Y 117.598,Z 431.963,A -85,B 0,C 180,E1 -25933.83,E2 -25933.83} C_VEL
LIN {X 0,Y 120.406,Z 439.481,A -85,B 0,C 180,E1 -25940.5,E2 -25940.5} C_VEL
LIN {X 0,Y 125.502,Z 445.675,A -85,B 0,C 180,E1 -25946.614,E2 -25946.614} C_VEL
LIN {X 0,Y 132.206,Z 450.551,A -85,B 0,C 180,E1 -25952.113,E2 -25952.113} C_VEL
LIN {X 0,Y 140.345,Z 454.228,A -85,B 0,C 180,E1 -25956.935,E2 -25956.935} C_VEL
LIN {X 0,Y 149.72,Z 456.753,A -85,B 0,C 180,E1 -25961.084,E2 -25961.084} C_VEL
LIN {X 0,Y 154.141,Z 457.583,A -85,B 0,C 180,E1 -25963.15,E2 -25963.15} C_VEL
LIN {X 0,Y 143.131,Z 456.735,A -85,B 0,C 180,E1 -25967.436,E2 -25967.436} C_VEL
LIN {X 0,Y 135.485,Z 455.193,A -85,B 0,C 180,E1 -25971.499,E2 -25971.499} C_VEL
LIN {X 0,Y 128.34,Z 452.572,A -85,B 0,C 180,E1 -25976.793,E2 -25976.793} C_VEL
LIN {X 0,Y 122.762,Z 448.861,A -85,B 0,C 180,E1 -25982.738,E2 -25982.738} C_VEL
LIN {X 0,Y 118.838,Z 443.391,A -85,B 0,C 180,E1 -25990.454,E2 -25990.454} C_VEL
LIN {X 0,Y 116.131,Z 447.981,A -85,B 0,C 180,E1 -25994.193,E2 -25994.193} C_VEL
LIN {X 0,Y 113.929,Z 452.85,A -85,B 0,C 180,E1 -25999.331,E2 -25999.331} C_VEL
LIN {X 0,Y 112.777,Z 457.176,A -85,B 0,C 180,E1 -26005.619,E2 -26005.619} C_VEL
LIN {X 0,Y 112.819,Z 459.317,A -85,B 0,C 180,E1 -26009.996,E2 -26009.996} C_VEL
LIN {X 0,Y 112.509,Z 460.538,A -85,B 0,C 180,E1 -26013.577,E2 -26013.577} C_VEL
LIN {X 0,Y 112.443,Z 461.361,A -85,B 0,C 180,E1 -26017.177,E2 -26017.177} C_VEL
LIN {X 0,Y 112.792,Z 461.778,A -85,B 0,C 180,E1 -26020.77,E2 -26020.77} C_VEL
LIN {X 0,Y 114.662,Z 461.407,A -85,B 0,C 180,E1 -26027.842,E2 -26027.842} C_VEL
LIN {X 0,Y 116.255,Z 460.659,A -85,B 0,C 180,E1 -26031.263,E2 -26031.263} C_VEL
LIN {X 0,Y 118.341,Z 459.509,A -85,B 0,C 180,E1 -26034.56,E2 -26034.56} C_VEL
LIN {X 0,Y 120.753,Z 457.927,A -85,B 0,C 180,E1 -26037.746,E2 -26037.746} C_VEL
LIN {X 0,Y 125.484,Z 454.449,A -85,B 0,C 180,E1 -26042.654,E2 -26042.654} C_VEL
LIN {X 0,Y 131.947,Z 448.987,A -85,B 0,C 180,E1 -26047.769,E2 -26047.769} C_VEL
LIN {X 0,Y 139.079,Z 442.111,A -85,B 0,C 180,E1 -26052.028,E2 -26052.028} C_VEL
LIN {X 0,Y 140.09,Z 441.072,A -85,B 0,C 180,E1 -26052.564,E2 -26052.564} C_VEL
LIN {X 0,Y 142.678,Z 437.867,A -85,B 0,C 180,E1 -26054.291,E2 -26054.291} C_VEL
LIN {X 0,Y 145.646,Z 432.298,A -85,B 0,C 180,E1 -26057.346,E2 -26057.346} C_VEL
LIN {X 0,Y 148.678,Z 426.109,A -85,B 0,C 180,E1 -26060.121,E2 -26060.121} C_VEL
LIN {X 0,Y 151.251,Z 421.936,A -85,B 0,C 180,E1 -26061.376,E2 -26061.376} C_VEL
LIN {X 0,Y 157.508,Z 412.214,A -85,B 0,C 180,E1 -26063.428,E2 -26063.428} C_VEL
LIN {X 0,Y 163.78,Z 400.725,A -85,B 0,C 180,E1 -26065.148,E2 -26065.148} C_VEL
LIN {X 0,Y 168.805,Z 389.278,A -85,B 0,C 180,E1 -26066.37,E2 -26066.37} C_VEL
LIN {X 0,Y 172.876,Z 377.081,A -85,B 0,C 180,E1 -26067.339,E2 -26067.339} C_VEL
LIN {X 0,Y 175.989,Z 364.029,A -85,B 0,C 180,E1 -26068.067,E2 -26068.067} C_VEL
LIN {X 0,Y 177.902,Z 349.79,A -85,B 0,C 180,E1 -26068.597,E2 -26068.597} C_VEL
LIN {X 0,Y 178.82,Z 339.436,A -85,B 0,C 180,E1 -26068.947,E2 -26068.947} C_VEL
LIN {X 0,Y 175.615,Z 332.898,A -85,B 0,C 180,E1 -26072.026,E2 -26072.026} C_VEL
LIN {X 0,Y 172.613,Z 327.19,A -85,B 0,C 180,E1 -26075.423,E2 -26075.423} C_VEL
LIN {X 0,Y 170.61,Z 323.637,A -85,B 0,C 180,E1 -26078.121,E2 -26078.121} C_VEL
LIN {X 0,Y 168.969,Z 320.675,A -85,B 0,C 180,E1 -26080.88,E2 -26080.88} C_VEL
LIN {X 0,Y 166.884,Z 316.731,A -85,B 0,C 180,E1 -26085.888,E2 -26085.888} C_VEL
LIN {X 0,Y 165.652,Z 315.294,A -85,B 0,C 180,E1 -26092.688,E2 -26092.688} C_VEL
LIN {X 0,Y 166.374,Z 315.791,A -85,B 0,C 180,E1 -26098.639,E2 -26098.639} C_VEL
LIN {X 0,Y 167.157,Z 316.775,A -85,B 0,C 180,E1 -26101.205,E2 -26101.205} C_VEL
LIN {X 0,Y 169.393,Z 321.15,A -85,B 0,C 180,E1 -26106.227,E2 -26106.227} C_VEL
LIN {X 0,Y 171.787,Z 325.607,A -85,B 0,C 180,E1 -26109.91,E2 -26109.91} C_VEL
LIN {X 0,Y 174.571,Z 330.596,A -85,B 0,C 180,E1 -26113.228,E2 -26113.228} C_VEL
LIN {X 0,Y 178.384,Z 338.353,A -85,B 0,C 180,E1 -26117.036,E2 -26117.036} C_VEL
LIN {X 0,Y 179.008,Z 339.795,A -85,B 0,C 180,E1 -26117.608,E2 -26117.608} C_VEL
LIN {X 0,Y 177.213,Z 354.884,A -85,B 0,C 180,E1 -26118.173,E2 -26118.173} C_VEL
LIN {X 0,Y 174.536,Z 367.678,A -85,B 0,C 180,E1 -26118.924,E2 -26118.924} C_VEL
LIN {X 0,Y 170.986,Z 379.432,A -85,B 0,C 180,E1 -26119.919,E2 -26119.919} C_VEL
LIN {X 0,Y 166.733,Z 390.292,A -85,B 0,C 180,E1 -26121.165,E2 -26121.165} C_VEL
LIN {X 0,Y 161.169,Z 401.683,A -85,B 0,C 180,E1 -26122.908,E2 -26122.908} C_VEL
LIN {X 0,Y 155.044,Z 411.841,A -85,B 0,C 180,E1 -26124.971,E2 -26124.971} C_VEL
LIN {X 0,Y 148.462,Z 420.947,A -85,B 0,C 180,E1 -26127.434,E2 -26127.434} C_VEL
LIN {X 0,Y 142.182,Z 428.447,A -85,B 0,C 180,E1 -26130.166,E2 -26130.166} C_VEL
LIN {X 0,Y 135.149,Z 435.661,A -85,B 0,C 180,E1 -26133.699,E2 -26133.699} C_VEL
LIN {X 0,Y 128.663,Z 441.349,A -85,B 0,C 180,E1 -26137.63,E2 -26137.63} C_VEL
LIN {X 0,Y 122.811,Z 445.742,A -85,B 0,C 180,E1 -26141.937,E2 -26141.937} C_VEL
LIN {X 0,Y 119.313,Z 448.03,A -85,B 0,C 180,E1 -26145.027,E2 -26145.027} C_VEL
LIN {X 0,Y 116.126,Z 449.842,A -85,B 0,C 180,E1 -26148.267,E2 -26148.267} C_VEL
LIN {X 0,Y 113.34,Z 451.166,A -85,B 0,C 180,E1 -26151.683,E2 -26151.683} C_VEL
LIN {X 0,Y 110.716,Z 452.153,A -85,B 0,C 180,E1 -26155.612,E2 -26155.612} C_VEL
LIN {X 0,Y 108.955,Z 452.557,A -85,B 0,C 180,E1 -26158.939,E2 -26158.939} C_VEL
LIN {X 0,Y 107.371,Z 452.578,A -85,B 0,C 180,E1 -26162.735,E2 -26162.735} C_VEL
LIN {X 0,Y 105.831,Z 451.884,A -85,B 0,C 180,E1 -26168.392,E2 -26168.392} C_VEL
LIN {X 0,Y 104.986,Z 450.166,A -85,B 0,C 180,E1 -26174.473,E2 -26174.473} C_VEL
LIN {X 0,Y 105.119,Z 447.503,A -85,B 0,C 180,E1 -26180.383,E2 -26180.383} C_VEL
LIN {X 0,Y 106.044,Z 443.803,A -85,B 0,C 180,E1 -26186.204,E2 -26186.204} C_VEL
LIN {X 0,Y 107.575,Z 438.992,A -85,B 0,C 180,E1 -26191.876,E2 -26191.876} C_VEL
LIN {X 0,Y 109.784,Z 432.929,A -85,B 0,C 180,E1 -26197.36,E2 -26197.36} C_VEL
LIN {X 0,Y 112.869,Z 425.37,A -85,B 0,C 180,E1 -26202.592,E2 -26202.592} C_VEL
LIN {X 0,Y 116.769,Z 415.836,A -85,B 0,C 180,E1 -26207.518,E2 -26207.518} C_VEL
LIN {X 0,Y 120.51,Z 406.125,A -85,B 0,C 180,E1 -26211.333,E2 -26211.333} C_VEL
LIN {X 0,Y 124.372,Z 394.913,A -85,B 0,C 180,E1 -26214.633,E2 -26214.633} C_VEL
LIN {X 0,Y 127.533,Z 384.09,A -85,B 0,C 180,E1 -26217.045,E2 -26217.045} C_VEL
LIN {X 0,Y 130.326,Z 371.26,A -85,B 0,C 180,E1 -26219.225,E2 -26219.225} C_VEL
LIN {X 0,Y 132.725,Z 357.95,A -85,B 0,C 180,E1 -26220.677,E2 -26220.677} C_VEL
LIN {X 0,Y 134.156,Z 344.721,A -85,B 0,C 180,E1 -26221.596,E2 -26221.596} C_VEL
LIN {X 0,Y 136.937,Z 303.869,A -85,B 0,C 180,E1 -26223.43,E2 -26223.43} C_VEL
LIN {X 0,Y 132.011,Z 293.046,A -85,B 0,C 180,E1 -26226.161,E2 -26226.161} C_VEL
LIN {X 0,Y 126.637,Z 283.182,A -85,B 0,C 180,E1 -26229.365,E2 -26229.365} C_VEL
LIN {X 0,Y 121.156,Z 274.662,A -85,B 0,C 180,E1 -26233.018,E2 -26233.018} C_VEL
LIN {X 0,Y 118.231,Z 270.612,A -85,B 0,C 180,E1 -26235.191,E2 -26235.191} C_VEL
LIN {X 0,Y 115.715,Z 266.963,A -85,B 0,C 180,E1 -26237.264,E2 -26237.264} C_VEL
LIN {X 0,Y 112.883,Z 263.649,A -85,B 0,C 180,E1 -26239.762,E2 -26239.762} C_VEL
LIN {X 0,Y 111.903,Z 261.647,A -85,B 0,C 180,E1 -26240.803,E2 -26240.803} C_VEL
LIN {X 0,Y 109.26,Z 259.639,A -85,B 0,C 180,E1 -26243.419,E2 -26243.419} C_VEL
LIN {X 0,Y 108.03,Z 257.364,A -85,B 0,C 180,E1 -26244.945,E2 -26244.945} C_VEL
LIN {X 0,Y 107.763,Z 256.055,A -85,B 0,C 180,E1 -26245.496,E2 -26245.496} C_VEL
LIN {X 0,Y 108.219,Z 255.96,A -85,B 0,C 180,E1 -26251.325,E2 -26251.325} C_VEL
LIN {X 0,Y 111.723,Z 272.317,A -85,B 0,C 180,E1 -26253.351,E2 -26253.351} C_VEL
LIN {X 0,Y 114.145,Z 282.008,A -85,B 0,C 180,E1 -26254.468,E2 -26254.468} C_VEL
LIN {X 0,Y 111.744,Z 347.981,A -85,B 0,C 180,E1 -26263.207,E2 -26263.207} C_VEL
LIN {X 0,Y 111.014,Z 362.634,A -85,B 0,C 180,E1 -26265.799,E2 -26265.799} C_VEL
LIN {X 0,Y 110.32,Z 375.99,A -85,B 0,C 180,E1 -26268.981,E2 -26268.981} C_VEL
LIN {X 0,Y 109.95,Z 386.72,A -85,B 0,C 180,E1 -26272.192,E2 -26272.192} C_VEL
LIN {X 0,Y 109.604,Z 398.987,A -85,B 0,C 180,E1 -26276.783,E2 -26276.783} C_VEL
LIN {X 0,Y 109.554,Z 407.952,A -85,B 0,C 180,E1 -26280.918,E2 -26280.918} C_VEL
LIN {X 0,Y 109.661,Z 414.749,A -85,B 0,C 180,E1 -26284.594,E2 -26284.594} C_VEL
LIN {X 0,Y 110.17,Z 423.19,A -85,B 0,C 180,E1 -26290.103,E2 -26290.103} C_VEL
LIN {X 0,Y 111.771,Z 431.305,A -85,B 0,C 180,E1 -26296.436,E2 -26296.436} C_VEL
LIN {X 0,Y 115.25,Z 438.908,A -85,B 0,C 180,E1 -26303.351,E2 -26303.351} C_VEL
LIN {X 0,Y 120.996,Z 445.259,A -85,B 0,C 180,E1 -26309.585,E2 -26309.585} C_VEL
LIN {X 0,Y 128.337,Z 450.31,A -85,B 0,C 180,E1 -26315.099,E2 -26315.099} C_VEL
LIN {X 0,Y 134.784,Z 453.287,A -85,B 0,C 180,E1 -26318.734,E2 -26318.734} C_VEL
LIN {X 0,Y 144.176,Z 456.274,A -85,B 0,C 180,E1 -26323.009,E2 -26323.009} C_VEL
LIN {X 0,Y 134.483,Z 454.629,A -85,B 0,C 180,E1 -26327.201,E2 -26327.201} C_VEL
LIN {X 0,Y 126.27,Z 452.09,A -85,B 0,C 180,E1 -26332.244,E2 -26332.244} C_VEL
LIN {X 0,Y 119.609,Z 448.564,A -85,B 0,C 180,E1 -26338.07,E2 -26338.07} C_VEL
LIN {X 0,Y 114.784,Z 443.95,A -85,B 0,C 180,E1 -26344.617,E2 -26344.617} C_VEL
LIN {X 0,Y 113.169,Z 441.247,A -85,B 0,C 180,E1 -26348.239,E2 -26348.239} C_VEL
LIN {X 0,Y 110.446,Z 445.347,A -85,B 0,C 180,E1 -26351.444,E2 -26351.444} C_VEL
LIN {X 0,Y 107.62,Z 450.703,A -85,B 0,C 180,E1 -26356.783,E2 -26356.783} C_VEL
LIN {X 0,Y 106.1,Z 454.898,A -85,B 0,C 180,E1 -26362.383,E2 -26362.383} C_VEL
LIN {X 0,Y 105.654,Z 457.109,A -85,B 0,C 180,E1 -26366.182,E2 -26366.182} C_VEL
LIN {X 0,Y 105.734,Z 458.85,A -85,B 0,C 180,E1 -26369.996,E2 -26369.996} C_VEL
LIN {X 0,Y 105.406,Z 460.103,A -85,B 0,C 180,E1 -26373.819,E2 -26373.819} C_VEL
LIN {X 0,Y 105.803,Z 461.434,A -85,B 0,C 180,E1 -26381.49,E2 -26381.49} C_VEL
LIN {X 0,Y 107.884,Z 461.142,A -85,B 0,C 180,E1 -26389.005,E2 -26389.005} C_VEL
LIN {X 0,Y 111.895,Z 459.336,A -85,B 0,C 180,E1 -26396.078,E2 -26396.078} C_VEL
LIN {X 0,Y 114.5,Z 457.802,A -85,B 0,C 180,E1 -26399.404,E2 -26399.404} C_VEL
LIN {X 0,Y 120.091,Z 453.99,A -85,B 0,C 180,E1 -26404.985,E2 -26404.985} C_VEL
LIN {X 0,Y 126.405,Z 449.031,A -85,B 0,C 180,E1 -26409.742,E2 -26409.742} C_VEL
LIN {X 0,Y 133.904,Z 442.291,A -85,B 0,C 180,E1 -26414.057,E2 -26414.057} C_VEL
LIN {X 0,Y 140.872,Z 434.991,A -85,B 0,C 180,E1 -26417.375,E2 -26417.375} C_VEL
LIN {X 0,Y 148.372,Z 425.936,A -85,B 0,C 180,E1 -26420.324,E2 -26420.324} C_VEL
LIN {X 0,Y 151.251,Z 421.936,A -85,B 0,C 180,E1 -26421.376,E2 -26421.376} C_VEL
LIN {X 0,Y 153.817,Z 417.64,A -85,B 0,C 180,E1 -26422.553,E2 -26422.553} C_VEL
LIN {X 0,Y 156.8,Z 410.41,A -85,B 0,C 180,E1 -26424.821,E2 -26424.821} C_VEL
LIN {X 0,Y 159.623,Z 402.8,A -85,B 0,C 180,E1 -26426.865,E2 -26426.865} C_VEL
LIN {X 0,Y 161.79,Z 397.823,A -85,B 0,C 180,E1 -26427.674,E2 -26427.674} C_VEL
LIN {X 0,Y 167.011,Z 385.446,A -85,B 0,C 180,E1 -26428.875,E2 -26428.875} C_VEL
LIN {X 0,Y 170.89,Z 373.104,A -85,B 0,C 180,E1 -26429.723,E2 -26429.723} C_VEL
LIN {X 0,Y 173.831,Z 359.223,A -85,B 0,C 180,E1 -26430.381,E2 -26430.381} C_VEL
LIN {X 0,Y 175.59,Z 343.212,A -85,B 0,C 180,E1 -26430.938,E2 -26430.938} C_VEL
LIN {X 0,Y 172.607,Z 336.816,A -85,B 0,C 180,E1 -26434.2,E2 -26434.2} C_VEL
LIN {X 0,Y 169.584,Z 330.899,A -85,B 0,C 180,E1 -26438.227,E2 -26438.227} C_VEL
LIN {X 0,Y 167.621,Z 327.34,A -85,B 0,C 180,E1 -26441.672,E2 -26441.672} C_VEL
LIN {X 0,Y 165.811,Z 323.658,A -85,B 0,C 180,E1 -26446.437,E2 -26446.437} C_VEL
LIN {X 0,Y 164.774,Z 322.345,A -85,B 0,C 180,E1 -26452.649,E2 -26452.649} C_VEL
LIN {X 0,Y 165.485,Z 322.87,A -85,B 0,C 180,E1 -26458.632,E2 -26458.632} C_VEL
LIN {X 0,Y 166.101,Z 323.721,A -85,B 0,C 180,E1 -26460.758,E2 -26460.758} C_VEL
LIN {X 0,Y 168.006,Z 327.685,A -85,B 0,C 180,E1 -26465.401,E2 -26465.401} C_VEL
LIN {X 0,Y 170.209,Z 332.098,A -85,B 0,C 180,E1 -26469.1,E2 -26469.1} C_VEL
LIN {X 0,Y 172.695,Z 336.831,A -85,B 0,C 180,E1 -26472.282,E2 -26472.282} C_VEL
LIN {X 0,Y 175.765,Z 343.415,A -85,B 0,C 180,E1 -26475.612,E2 -26475.612} C_VEL
LIN {X 0,Y 173.787,Z 357.798,A -85,B 0,C 180,E1 -26476.189,E2 -26476.189} C_VEL
LIN {X 0,Y 171.019,Z 369.641,A -85,B 0,C 180,E1 -26476.922,E2 -26476.922} C_VEL
LIN {X 0,Y 167.136,Z 381.59,A -85,B 0,C 180,E1 -26477.951,E2 -26477.951} C_VEL
LIN {X 0,Y 162.761,Z 392.089,A -85,B 0,C 180,E1 -26479.178,E2 -26479.178} C_VEL
LIN {X 0,Y 157.095,Z 403.038,A -85,B 0,C 180,E1 -26480.862,E2 -26480.862} C_VEL
LIN {X 0,Y 150.695,Z 413.078,A -85,B 0,C 180,E1 -26482.923,E2 -26482.923} C_VEL
LIN {X 0,Y 143.868,Z 422.03,A -85,B 0,C 180,E1 -26485.355,E2 -26485.355} C_VEL
LIN {X 0,Y 137.168,Z 429.598,A -85,B 0,C 180,E1 -26488.17,E2 -26488.17} C_VEL
LIN {X 0,Y 129.991,Z 436.458,A -85,B 0,C 180,E1 -26491.629,E2 -26491.629} C_VEL
LIN {X 0,Y 123.913,Z 441.491,A -85,B 0,C 180,E1 -26495.132,E2 -26495.132} C_VEL
LIN {X 0,Y 117.974,Z 445.729,A -85,B 0,C 180,E1 -26499.252,E2 -26499.252} C_VEL
LIN {X 0,Y 113.634,Z 448.382,A -85,B 0,C 180,E1 -26502.871,E2 -26502.871} C_VEL
LIN {X 0,Y 110.695,Z 449.95,A -85,B 0,C 180,E1 -26505.708,E2 -26505.708} C_VEL
LIN {X 0,Y 107.605,Z 451.338,A -85,B 0,C 180,E1 -26509.228,E2 -26509.228} C_VEL
LIN {X 0,Y 104.305,Z 452.494,A -85,B 0,C 180,E1 -26513.956,E2 -26513.956} C_VEL
LIN {X 0,Y 100.847,Z 452.927,A -85,B 0,C 180,E1 -26520.807,E2 -26520.807} C_VEL
LIN {X 0,Y 98.859,Z 452.173,A -85,B 0,C 180,E1 -26527.549,E2 -26527.549} C_VEL
LIN {X 0,Y 97.962,Z 450.693,A -85,B 0,C 180,E1 -26533.328,E2 -26533.328} C_VEL
LIN {X 0,Y 97.954,Z 448.122,A -85,B 0,C 180,E1 -26539.672,E2 -26539.672} C_VEL
LIN {X 0,Y 98.836,Z 444.518,A -85,B 0,C 180,E1 -26545.927,E2 -26545.927} C_VEL
LIN {X 0,Y 100.421,Z 439.805,A -85,B 0,C 180,E1 -26552.01,E2 -26552.01} C_VEL
LIN {X 0,Y 102.722,Z 433.854,A -85,B 0,C 180,E1 -26557.869,E2 -26557.869} C_VEL
LIN {X 0,Y 105.934,Z 426.432,A -85,B 0,C 180,E1 -26563.431,E2 -26563.431} C_VEL
LIN {X 0,Y 109.285,Z 418.84,A -85,B 0,C 180,E1 -26567.79,E2 -26567.79} C_VEL
LIN {X 0,Y 113.099,Z 409.596,A -85,B 0,C 180,E1 -26571.895,E2 -26571.895} C_VEL
LIN {X 0,Y 116.992,Z 399.337,A -85,B 0,C 180,E1 -26575.346,E2 -26575.346} C_VEL
LIN {X 0,Y 120.32,Z 389.496,A -85,B 0,C 180,E1 -26577.862,E2 -26577.862} C_VEL
LIN {X 0,Y 123.106,Z 379.078,A -85,B 0,C 180,E1 -26579.973,E2 -26579.973} C_VEL
LIN {X 0,Y 125.448,Z 368.288,A -85,B 0,C 180,E1 -26581.612,E2 -26581.612} C_VEL
LIN {X 0,Y 127.584,Z 355.766,A -85,B 0,C 180,E1 -26582.894,E2 -26582.894} C_VEL
LIN {X 0,Y 128.975,Z 342.1,A -85,B 0,C 180,E1 -26583.742,E2 -26583.742} C_VEL
LIN {X 0,Y 131.579,Z 306.237,A -85,B 0,C 180,E1 -26585.355,E2 -26585.355} C_VEL
LIN {X 0,Y 127.69,Z 297.475,A -85,B 0,C 180,E1 -26587.705,E2 -26587.705} C_VEL
LIN {X 0,Y 122.962,Z 288.459,A -85,B 0,C 180,E1 -26590.774,E2 -26590.774} C_VEL
LIN {X 0,Y 117.882,Z 280.221,A -85,B 0,C 180,E1 -26594.456,E2 -26594.456} C_VEL
LIN {X 0,Y 114.824,Z 275.913,A -85,B 0,C 180,E1 -26596.93,E2 -26596.93} C_VEL
LIN {X 0,Y 112.204,Z 272.149,A -85,B 0,C 180,E1 -26599.302,E2 -26599.302} C_VEL
LIN {X 0,Y 109.769,Z 268.759,A -85,B 0,C 180,E1 -26601.75,E2 -26601.75} C_VEL
LIN {X 0,Y 108.958,Z 267.716,A -85,B 0,C 180,E1 -26602.62,E2 -26602.62} C_VEL
LIN {X 0,Y 106.383,Z 264.977,A -85,B 0,C 180,E1 -26605.55,E2 -26605.55} C_VEL
LIN {X 0,Y 105.364,Z 262.691,A -85,B 0,C 180,E1 -26607.021,E2 -26607.021} C_VEL
LIN {X 0,Y 103.386,Z 261.579,A -85,B 0,C 180,E1 -26609.628,E2 -26609.628} C_VEL
LIN {X 0,Y 102.808,Z 262.186,A -85,B 0,C 180,E1 -26610.289,E2 -26610.289} C_VEL
LIN {X 0,Y 102.104,Z 261.748,A -85,B 0,C 180,E1 -26611.358,E2 -26611.358} C_VEL
LIN {X 0,Y 101.794,Z 260.481,A -85,B 0,C 180,E1 -26612.064,E2 -26612.064} C_VEL
LIN {X 0,Y 105.874,Z 277.551,A -85,B 0,C 180,E1 -26614.274,E2 -26614.274} C_VEL
LIN {X 0,Y 107.019,Z 282.72,A -85,B 0,C 180,E1 -26614.9,E2 -26614.9} C_VEL
LIN {X 0,Y 104.872,Z 347.763,A -85,B 0,C 180,E1 -26624.201,E2 -26624.201} C_VEL
LIN {X 0,Y 104.248,Z 361.832,A -85,B 0,C 180,E1 -26626.847,E2 -26626.847} C_VEL
LIN {X 0,Y 103.646,Z 375.231,A -85,B 0,C 180,E1 -26630.239,E2 -26630.239} C_VEL
LIN {X 0,Y 103.343,Z 386.007,A -85,B 0,C 180,E1 -26633.654,E2 -26633.654} C_VEL
LIN {X 0,Y 103.147,Z 397.2,A -85,B 0,C 180,E1 -26638.047,E2 -26638.047} C_VEL
LIN {X 0,Y 103.188,Z 405.399,A -85,B 0,C 180,E1 -26641.951,E2 -26641.951} C_VEL
LIN {X 0,Y 103.403,Z 412.371,A -85,B 0,C 180,E1 -26645.851,E2 -26645.851} C_VEL
LIN {X 0,Y 104.055,Z 421.071,A -85,B 0,C 180,E1 -26651.69,E2 -26651.69} C_VEL
LIN {X 0,Y 105.881,Z 429.439,A -85,B 0,C 180,E1 -26658.377,E2 -26658.377} C_VEL
LIN {X 0,Y 109.666,Z 437.197,A -85,B 0,C 180,E1 -26665.437,E2 -26665.437} C_VEL
LIN {X 0,Y 115.258,Z 443.379,A -85,B 0,C 180,E1 -26671.38,E2 -26671.38} C_VEL
LIN {X 0,Y 122.742,Z 448.758,A -85,B 0,C 180,E1 -26676.956,E2 -26676.956} C_VEL
LIN {X 0,Y 129.397,Z 452.088,A -85,B 0,C 180,E1 -26680.674,E2 -26680.674} C_VEL
LIN {X 0,Y 134.209,Z 453.975,A -85,B 0,C 180,E1 -26682.902,E2 -26682.902} C_VEL
LIN {X 0,Y 125.058,Z 451.514,A -85,B 0,C 180,E1 -26687.59,E2 -26687.59} C_VEL
LIN {X 0,Y 117.303,Z 448.114,A -85,B 0,C 180,E1 -26693.188,E2 -26693.188} C_VEL
LIN {X 0,Y 111.208,Z 443.675,A -85,B 0,C 180,E1 -26699.626,E2 -26699.626} C_VEL
LIN {X 0,Y 107.624,Z 439.095,A -85,B 0,C 180,E1 -26705.908,E2 -26705.908} C_VEL
LIN {X 0,Y 103.793,Z 444.613,A -85,B 0,C 180,E1 -26710.206,E2 -26710.206} C_VEL
LIN {X 0,Y 100.757,Z 450.052,A -85,B 0,C 180,E1 -26715.865,E2 -26715.865} C_VEL
LIN {X 0,Y 99.075,Z 454.322,A -85,B 0,C 180,E1 -26721.839,E2 -26721.839} C_VEL
LIN {X 0,Y 98.545,Z 457.014,A -85,B 0,C 180,E1 -26726.794,E2 -26726.794} C_VEL
LIN {X 0,Y 98.648,Z 458.381,A -85,B 0,C 180,E1 -26729.995,E2 -26729.995} C_VEL
LIN {X 0,Y 98.31,Z 459.669,A -85,B 0,C 180,E1 -26734.095,E2 -26734.095} C_VEL
LIN {X 0,Y 98.843,Z 461.071,A -85,B 0,C 180,E1 -26742.312,E2 -26742.312} C_VEL
LIN {X 0,Y 99.774,Z 461.183,A -85,B 0,C 180,E1 -26746.36,E2 -26746.36} C_VEL
LIN {X 0,Y 103.129,Z 460.2,A -85,B 0,C 180,E1 -26754.13,E2 -26754.13} C_VEL
LIN {X 0,Y 105.529,Z 459.144,A -85,B 0,C 180,E1 -26757.782,E2 -26757.782} C_VEL
LIN {X 0,Y 108.357,Z 457.683,A -85,B 0,C 180,E1 -26761.252,E2 -26761.252} C_VEL
LIN {X 0,Y 113.818,Z 454.301,A -85,B 0,C 180,E1 -26766.61,E2 -26766.61} C_VEL
LIN {X 0,Y 121.015,Z 449.08,A -85,B 0,C 180,E1 -26771.898,E2 -26771.898} C_VEL
LIN {X 0,Y 127.718,Z 443.532,A -85,B 0,C 180,E1 -26775.667,E2 -26775.667} C_VEL
LIN {X 0,Y 134.962,Z 436.62,A -85,B 0,C 180,E1 -26779.026,E2 -26779.026} C_VEL
LIN {X 0,Y 142.614,Z 427.991,A -85,B 0,C 180,E1 -26782.038,E2 -26782.038} C_VEL
LIN {X 0,Y 149.305,Z 419.172,A -85,B 0,C 180,E1 -26784.285,E2 -26784.285} C_VEL
LIN {X 0,Y 155.538,Z 409.499,A -85,B 0,C 180,E1 -26786.122,E2 -26786.122} C_VEL
LIN {X 0,Y 161.325,Z 398.802,A -85,B 0,C 180,E1 -26787.565,E2 -26787.565} C_VEL
LIN {X 0,Y 161.79,Z 397.823,A -85,B 0,C 180,E1 -26787.674,E2 -26787.674} C_VEL
LIN {X 0,Y 163.84,Z 392.711,A -85,B 0,C 180,E1 -26788.417,E2 -26788.417} C_VEL
LIN {X 0,Y 165.957,Z 384.229,A -85,B 0,C 180,E1 -26790.073,E2 -26790.073} C_VEL
LIN {X 0,Y 167.638,Z 375.502,A -85,B 0,C 180,E1 -26791.58,E2 -26791.58} C_VEL
LIN {X 0,Y 168.892,Z 369.944,A -85,B 0,C 180,E1 -26792.097,E2 -26792.097} C_VEL
LIN {X 0,Y 171.468,Z 356.962,A -85,B 0,C 180,E1 -26792.646,E2 -26792.646} C_VEL
LIN {X 0,Y 172.586,Z 347.08,A -85,B 0,C 180,E1 -26792.984,E2 -26792.984} C_VEL
LIN {X 0,Y 169.584,Z 340.466,A -85,B 0,C 180,E1 -26796.782,E2 -26796.782} C_VEL
LIN {X 0,Y 167.592,Z 336.511,A -85,B 0,C 180,E1 -26799.92,E2 -26799.92} C_VEL
LIN {X 0,Y 166.452,Z 334.19,A -85,B 0,C 180,E1 -26802.175,E2 -26802.175} C_VEL
LIN {X 0,Y 164.738,Z 330.549,A -85,B 0,C 180,E1 -26807.058,E2 -26807.058} C_VEL
LIN {X 0,Y 163.898,Z 329.389,A -85,B 0,C 180,E1 -26812.609,E2 -26812.609} C_VEL
LIN {X 0,Y 164.597,Z 329.947,A -85,B 0,C 180,E1 -26818.624,E2 -26818.624} C_VEL
LIN {X 0,Y 165.097,Z 330.78,A -85,B 0,C 180,E1 -26820.458,E2 -26820.458} C_VEL
LIN {X 0,Y 166.776,Z 334.547,A -85,B 0,C 180,E1 -26824.835,E2 -26824.835} C_VEL
LIN {X 0,Y 168.753,Z 338.731,A -85,B 0,C 180,E1 -26828.382,E2 -26828.382} C_VEL
LIN {X 0,Y 170.995,Z 343.375,A -85,B 0,C 180,E1 -26831.484,E2 -26831.484} C_VEL
LIN {X 0,Y 172.677,Z 347.228,A -85,B 0,C 180,E1 -26833.533,E2 -26833.533} C_VEL
LIN {X 0,Y 170.588,Z 360.277,A -85,B 0,C 180,E1 -26834.136,E2 -26834.136} C_VEL
LIN {X 0,Y 167.291,Z 372.992,A -85,B 0,C 180,E1 -26834.941,E2 -26834.941} C_VEL
LIN {X 0,Y 163.501,Z 383.758,A -85,B 0,C 180,E1 -26835.904,E2 -26835.904} C_VEL
LIN {X 0,Y 159.001,Z 393.874,A -85,B 0,C 180,E1 -26837.1,E2 -26837.1} C_VEL
LIN {X 0,Y 153.129,Z 404.496,A -85,B 0,C 180,E1 -26838.741,E2 -26838.741} C_VEL
LIN {X 0,Y 146.538,Z 414.312,A -85,B 0,C 180,E1 -26840.744,E2 -26840.744} C_VEL
LIN {X 0,Y 139.481,Z 423.113,A -85,B 0,C 180,E1 -26843.147,E2 -26843.147} C_VEL
LIN {X 0,Y 131.416,Z 431.55,A -85,B 0,C 180,E1 -26846.4,E2 -26846.4} C_VEL
LIN {X 0,Y 123.77,Z 438.269,A -85,B 0,C 180,E1 -26850.018,E2 -26850.018} C_VEL
LIN {X 0,Y 117.858,Z 442.743,A -85,B 0,C 180,E1 -26853.409,E2 -26853.409} C_VEL
LIN {X 0,Y 111.329,Z 446.959,A -85,B 0,C 180,E1 -26857.905,E2 -26857.905} C_VEL
LIN {X 0,Y 105.52,Z 450.033,A -85,B 0,C 180,E1 -26862.898,E2 -26862.898} C_VEL
LIN {X 0,Y 102.11,Z 451.51,A -85,B 0,C 180,E1 -26866.512,E2 -26866.512} C_VEL
LIN {X 0,Y 97.915,Z 452.847,A -85,B 0,C 180,E1 -26872.145,E2 -26872.145} C_VEL
LIN {X 0,Y 94.454,Z 453.272,A -85,B 0,C 180,E1 -26878.617,E2 -26878.617} C_VEL
LIN {X 0,Y 91.927,Z 452.462,A -85,B 0,C 180,E1 -26886.555,E2 -26886.555} C_VEL
LIN {X 0,Y 90.992,Z 451.196,A -85,B 0,C 180,E1 -26892.009,E2 -26892.009} C_VEL
LIN {X 0,Y 90.737,Z 449.636,A -85,B 0,C 180,E1 -26896.569,E2 -26896.569} C_VEL
LIN {X 0,Y 91.25,Z 446.476,A -85,B 0,C 180,E1 -26903.371,E2 -26903.371} C_VEL
LIN {X 0,Y 92.632,Z 442.245,A -85,B 0,C 180,E1 -26910.005,E2 -26910.005} C_VEL
LIN {X 0,Y 95.251,Z 435.832,A -85,B 0,C 180,E1 -26917.424,E2 -26917.424} C_VEL
LIN {X 0,Y 98.443,Z 428.8,A -85,B 0,C 180,E1 -26923.421,E2 -26923.421} C_VEL
LIN {X 0,Y 102.541,Z 420.009,A -85,B 0,C 180,E1 -26929.004,E2 -26929.004} C_VEL
LIN {X 0,Y 106.536,Z 410.999,A -85,B 0,C 180,E1 -26933.321,E2 -26933.321} C_VEL
LIN {X 0,Y 110.714,Z 400.751,A -85,B 0,C 180,E1 -26936.989,E2 -26936.989} C_VEL
LIN {X 0,Y 114.591,Z 389.897,A -85,B 0,C 180,E1 -26939.893,E2 -26939.893} C_VEL
LIN {X 0,Y 117.536,Z 379.493,A -85,B 0,C 180,E1 -26942.055,E2 -26942.055} C_VEL
LIN {X 0,Y 120.092,Z 368.328,A -85,B 0,C 180,E1 -26943.781,E2 -26943.781} C_VEL
LIN {X 0,Y 122.318,Z 355.714,A -85,B 0,C 180,E1 -26945.074,E2 -26945.074} C_VEL
LIN {X 0,Y 123.774,Z 342.009,A -85,B 0,C 180,E1 -26945.916,E2 -26945.916} C_VEL
LIN {X 0,Y 126.31,Z 308.37,A -85,B 0,C 180,E1 -26947.463,E2 -26947.463} C_VEL
LIN {X 0,Y 122.552,Z 299.932,A -85,B 0,C 180,E1 -26949.988,E2 -26949.988} C_VEL
LIN {X 0,Y 117.974,Z 291.242,A -85,B 0,C 180,E1 -26953.325,E2 -26953.325} C_VEL
LIN {X 0,Y 113.983,Z 284.765,A -85,B 0,C 180,E1 -26956.57,E2 -26956.57} C_VEL
LIN {X 0,Y 111.276,Z 280.775,A -85,B 0,C 180,E1 -26959.023,E2 -26959.023} C_VEL
LIN {X 0,Y 109.461,Z 278.045,A -85,B 0,C 180,E1 -26960.843,E2 -26960.843} C_VEL
LIN {X 0,Y 106.673,Z 274.045,A -85,B 0,C 180,E1 -26963.949,E2 -26963.949} C_VEL
LIN {X 0,Y 104.016,Z 270.869,A -85,B 0,C 180,E1 -26967.279,E2 -26967.279} C_VEL
LIN {X 0,Y 103.238,Z 269.232,A -85,B 0,C 180,E1 -26968.489,E2 -26968.489} C_VEL
LIN {X 0,Y 102.712,Z 268.994,A -85,B 0,C 180,E1 -26969.197,E2 -26969.197} C_VEL
LIN {X 0,Y 101.039,Z 274.605,A -85,B 0,C 180,E1 -26970.419,E2 -26970.419} C_VEL
LIN {X 0,Y 99.818,Z 277.205,A -85,B 0,C 180,E1 -26971.68,E2 -26971.68} C_VEL
LIN {X 0,Y 99.081,Z 277.916,A -85,B 0,C 180,E1 -26972.673,E2 -26972.673} C_VEL
LIN {X 0,Y 98.566,Z 277.536,A -85,B 0,C 180,E1 -26973.599,E2 -26973.599} C_VEL
LIN {X 0,Y 98.293,Z 276.302,A -85,B 0,C 180,E1 -26974.544,E2 -26974.544} C_VEL
LIN {X 0,Y 99.945,Z 283.416,A -85,B 0,C 180,E1 -26975.46,E2 -26975.46} C_VEL
LIN {X 0,Y 98.088,Z 347.183,A -85,B 0,C 180,E1 -26985.343,E2 -26985.343} C_VEL
LIN {X 0,Y 97.569,Z 360.76,A -85,B 0,C 180,E1 -26988.047,E2 -26988.047} C_VEL
LIN {X 0,Y 97.065,Z 374.304,A -85,B 0,C 180,E1 -26991.673,E2 -26991.673} C_VEL
LIN {X 0,Y 96.855,Z 385.127,A -85,B 0,C 180,E1 -26995.317,E2 -26995.317} C_VEL
LIN {X 0,Y 96.842,Z 396.329,A -85,B 0,C 180,E1 -26999.999,E2 -26999.999} C_VEL
LIN {X 0,Y 97.121,Z 406.423,A -85,B 0,C 180,E1 -27005.189,E2 -27005.189} C_VEL
LIN {X 0,Y 97.562,Z 414.542,A -85,B 0,C 180,E1 -27010.374,E2 -27010.374} C_VEL
LIN {X 0,Y 99.15,Z 423.97,A -85,B 0,C 180,E1 -27017.532,E2 -27017.532} C_VEL
LIN {X 0,Y 102.049,Z 431.688,A -85,B 0,C 180,E1 -27024.406,E2 -27024.406} C_VEL
LIN {X 0,Y 107.713,Z 439.253,A -85,B 0,C 180,E1 -27031.464,E2 -27031.464} C_VEL
LIN {X 0,Y 115.188,Z 445.516,A -85,B 0,C 180,E1 -27037.598,E2 -27037.598} C_VEL
LIN {X 0,Y 124.212,Z 450.618,A -85,B 0,C 180,E1 -27042.762,E2 -27042.762} C_VEL
LIN {X 0,Y 120.174,Z 449.319,A -85,B 0,C 180,E1 -27045.425,E2 -27045.425} C_VEL
LIN {X 0,Y 112.083,Z 445.552,A -85,B 0,C 180,E1 -27051.163,E2 -27051.163} C_VEL
LIN {X 0,Y 105.698,Z 440.734,A -85,B 0,C 180,E1 -27057.859,E2 -27057.859} C_VEL
LIN {X 0,Y 102.455,Z 436.711,A -85,B 0,C 180,E1 -27063.242,E2 -27063.242} C_VEL
LIN {X 0,Y 97.854,Z 442.811,A -85,B 0,C 180,E1 -27067.843,E2 -27067.843} C_VEL
LIN {X 0,Y 94.837,Z 447.681,A -85,B 0,C 180,E1 -27072.752,E2 -27072.752} C_VEL
LIN {X 0,Y 92.551,Z 452.417,A -85,B 0,C 180,E1 -27079.052,E2 -27079.052} C_VEL
LIN {X 0,Y 91.549,Z 456.035,A -85,B 0,C 180,E1 -27085.592,E2 -27085.592} C_VEL
LIN {X 0,Y 91.552,Z 457.893,A -85,B 0,C 180,E1 -27089.995,E2 -27089.995} C_VEL
LIN {X 0,Y 91.215,Z 459.233,A -85,B 0,C 180,E1 -27094.414,E2 -27094.414} C_VEL
LIN {X 0,Y 91.881,Z 460.701,A -85,B 0,C 180,E1 -27103.261,E2 -27103.261} C_VEL
LIN {X 0,Y 92.948,Z 460.867,A -85,B 0,C 180,E1 -27107.6,E2 -27107.6} C_VEL
LIN {X 0,Y 94.5,Z 460.615,A -85,B 0,C 180,E1 -27111.825,E2 -27111.825} C_VEL
LIN {X 0,Y 99.27,Z 458.956,A -85,B 0,C 180,E1 -27119.703,E2 -27119.703} C_VEL
LIN {X 0,Y 102.34,Z 457.553,A -85,B 0,C 180,E1 -27123.319,E2 -27123.319} C_VEL
LIN {X 0,Y 107.75,Z 454.534,A -85,B 0,C 180,E1 -27128.492,E2 -27128.492} C_VEL
LIN {X 0,Y 113.632,Z 450.7,A -85,B 0,C 180,E1 -27132.865,E2 -27132.865} C_VEL
LIN {X 0,Y 120.439,Z 445.655,A -85,B 0,C 180,E1 -27136.832,E2 -27136.832} C_VEL
LIN {X 0,Y 127.824,Z 439.316,A -85,B 0,C 180,E1 -27140.325,E2 -27140.325} C_VEL
LIN {X 0,Y 135.69,Z 431.426,A -85,B 0,C 180,E1 -27143.394,E2 -27143.394} C_VEL
LIN {X 0,Y 142.489,Z 423.409,A -85,B 0,C 180,E1 -27145.701,E2 -27145.701} C_VEL
LIN {X 0,Y 149.522,Z 413.654,A -85,B 0,C 180,E1 -27147.779,E2 -27147.779} C_VEL
LIN {X 0,Y 156.154,Z 402.648,A -85,B 0,C 180,E1 -27149.395,E2 -27149.395} C_VEL
LIN {X 0,Y 162.148,Z 390.267,A -85,B 0,C 180,E1 -27150.692,E2 -27150.692} C_VEL
LIN {X 0,Y 166.601,Z 378.074,A -85,B 0,C 180,E1 -27151.628,E2 -27151.628} C_VEL
LIN {X 0,Y 168.892,Z 369.944,A -85,B 0,C 180,E1 -27152.097,E2 -27152.097} C_VEL
LIN {X 0,Y 169.997,Z 364.587,A -85,B 0,C 180,E1 -27152.464,E2 -27152.464} C_VEL
LIN {X 0,Y 170.478,Z 359.354,A -85,B 0,C 180,E1 -27153.088,E2 -27153.088} C_VEL
LIN {X 0,Y 170.358,Z 354.634,A -85,B 0,C 180,E1 -27154.002,E2 -27154.002} C_VEL
LIN {X 0,Y 169.763,Z 351.237,A -85,B 0,C 180,E1 -27155.094,E2 -27155.094} C_VEL
LIN {X 0,Y 169.638,Z 350.839,A -85,B 0,C 180,E1 -27155.275,E2 -27155.275} C_VEL
LIN {X 0,Y 167.525,Z 345.978,A -85,B 0,C 180,E1 -27158.367,E2 -27158.367} C_VEL
LIN {X 0,Y 165.915,Z 342.434,A -85,B 0,C 180,E1 -27161.317,E2 -27161.317} C_VEL
LIN {X 0,Y 165.093,Z 340.729,A -85,B 0,C 180,E1 -27163.142,E2 -27163.142} C_VEL
LIN {X 0,Y 163.704,Z 337.475,A -85,B 0,C 180,E1 -27167.605,E2 -27167.605} C_VEL
LIN {X 0,Y 163.02,Z 336.445,A -85,B 0,C 180,E1 -27172.569,E2 -27172.569} C_VEL
LIN {X 0,Y 163.71,Z 337.014,A -85,B 0,C 180,E1 -27178.617,E2 -27178.617} C_VEL
LIN {X 0,Y 164.06,Z 337.707,A -85,B 0,C 180,E1 -27180.001,E2 -27180.001} C_VEL
LIN {X 0,Y 165.566,Z 341.384,A -85,B 0,C 180,E1 -27184.261,E2 -27184.261} C_VEL
LIN {X 0,Y 167.253,Z 345.256,A -85,B 0,C 180,E1 -27187.546,E2 -27187.546} C_VEL
LIN {X 0,Y 169.096,Z 349.517,A -85,B 0,C 180,E1 -27190.477,E2 -27190.477} C_VEL
LIN {X 0,Y 169.723,Z 351.202,A -85,B 0,C 180,E1 -27191.42,E2 -27191.42} C_VEL
LIN {X 0,Y 167.909,Z 361.438,A -85,B 0,C 180,E1 -27191.945,E2 -27191.945} C_VEL
LIN {X 0,Y 164.349,Z 374.437,A -85,B 0,C 180,E1 -27192.75,E2 -27192.75} C_VEL
LIN {X 0,Y 160.071,Z 385.749,A -85,B 0,C 180,E1 -27193.747,E2 -27193.747} C_VEL
LIN {X 0,Y 154.689,Z 396.977,A -85,B 0,C 180,E1 -27195.116,E2 -27195.116} C_VEL
LIN {X 0,Y 149.106,Z 406.387,A -85,B 0,C 180,E1 -27196.582,E2 -27196.582} C_VEL
LIN {X 0,Y 142.609,Z 415.549,A -85,B 0,C 180,E1 -27198.448,E2 -27198.448} C_VEL
LIN {X 0,Y 135.307,Z 424.15,A -85,B 0,C 180,E1 -27200.791,E2 -27200.791} C_VEL
LIN {X 0,Y 126.929,Z 432.448,A -85,B 0,C 180,E1 -27204.002,E2 -27204.002} C_VEL
LIN {X 0,Y 118.948,Z 439.061,A -85,B 0,C 180,E1 -27207.6,E2 -27207.6} C_VEL
LIN {X 0,Y 111.535,Z 444.223,A -85,B 0,C 180,E1 -27211.725,E2 -27211.725} C_VEL
LIN {X 0,Y 104.732,Z 448.136,A -85,B 0,C 180,E1 -27216.373,E2 -27216.373} C_VEL
LIN {X 0,Y 100.603,Z 450.116,A -85,B 0,C 180,E1 -27219.793,E2 -27219.793} C_VEL
LIN {X 0,Y 96.854,Z 451.66,A -85,B 0,C 180,E1 -27223.486,E2 -27223.486} C_VEL
LIN {X 0,Y 91.681,Z 453.189,A -85,B 0,C 180,E1 -27230.049,E2 -27230.049} C_VEL
LIN {X 0,Y 88.215,Z 453.586,A -85,B 0,C 180,E1 -27236.11,E2 -27236.11} C_VEL
LIN {X 0,Y 86.323,Z 453.373,A -85,B 0,C 180,E1 -27240.764,E2 -27240.764} C_VEL
LIN {X 0,Y 84.981,Z 452.719,A -85,B 0,C 180,E1 -27245.581,E2 -27245.581} C_VEL
LIN {X 0,Y 84.062,Z 451.672,A -85,B 0,C 180,E1 -27250.468,E2 -27250.468} C_VEL
LIN {X 0,Y 83.65,Z 450.198,A -85,B 0,C 180,E1 -27255.407,E2 -27255.407} C_VEL
LIN {X 0,Y 84.066,Z 447.125,A -85,B 0,C 180,E1 -27262.801,E2 -27262.801} C_VEL
LIN {X 0,Y 85.457,Z 442.986,A -85,B 0,C 180,E1 -27270.005,E2 -27270.005} C_VEL
LIN {X 0,Y 88.153,Z 436.677,A -85,B 0,C 180,E1 -27278.025,E2 -27278.025} C_VEL
LIN {X 0,Y 91.515,Z 429.808,A -85,B 0,C 180,E1 -27284.458,E2 -27284.458} C_VEL
LIN {X 0,Y 95.823,Z 421.171,A -85,B 0,C 180,E1 -27290.393,E2 -27290.393} C_VEL
LIN {X 0,Y 100.541,Z 411.261,A -85,B 0,C 180,E1 -27295.41,E2 -27295.41} C_VEL
LIN {X 0,Y 104.85,Z 401.346,A -85,B 0,C 180,E1 -27299.084,E2 -27299.084} C_VEL
LIN {X 0,Y 109.02,Z 390.282,A -85,B 0,C 180,E1 -27302.134,E2 -27302.134} C_VEL
LIN {X 0,Y 112.153,Z 379.888,A -85,B 0,C 180,E1 -27304.336,E2 -27304.336} C_VEL
LIN {X 0,Y 114.827,Z 368.755,A -85,B 0,C 180,E1 -27306.098,E2 -27306.098} C_VEL
LIN {X 0,Y 117.203,Z 355.909,A -85,B 0,C 180,E1 -27307.427,E2 -27307.427} C_VEL
LIN {X 0,Y 118.813,Z 341.157,A -85,B 0,C 180,E1 -27308.319,E2 -27308.319} C_VEL
LIN {X 0,Y 121.235,Z 310.705,A -85,B 0,C 180,E1 -27309.73,E2 -27309.73} C_VEL
LIN {X 0,Y 116.753,Z 300.729,A -85,B 0,C 180,E1 -27313.144,E2 -27313.144} C_VEL
LIN {X 0,Y 112.601,Z 293.133,A -85,B 0,C 180,E1 -27316.64,E2 -27316.64} C_VEL
LIN {X 0,Y 108.955,Z 287.24,A -85,B 0,C 180,E1 -27320.13,E2 -27320.13} C_VEL
LIN {X 0,Y 106.479,Z 283.472,A -85,B 0,C 180,E1 -27322.83,E2 -27322.83} C_VEL
LIN {X 0,Y 104.288,Z 280.195,A -85,B 0,C 180,E1 -27325.52,E2 -27325.52} C_VEL
LIN {X 0,Y 103.163,Z 278.958,A -85,B 0,C 180,E1 -27326.974,E2 -27326.974} C_VEL
LIN {X 0,Y 102.715,Z 279.155,A -85,B 0,C 180,E1 -27327.47,E2 -27327.47} C_VEL
LIN {X 0,Y 100.957,Z 282.554,A -85,B 0,C 180,E1 -27329.08,E2 -27329.08} C_VEL
LIN {X 0,Y 99.353,Z 284.45,A -85,B 0,C 180,E1 -27330.932,E2 -27330.932} C_VEL
LIN {X 0,Y 98.984,Z 284.689,A -85,B 0,C 180,E1 -27331.427,E2 -27331.427} C_VEL
LIN {X 0,Y 95.385,Z 299.018,A -85,B 0,C 180,E1 -27334.203,E2 -27334.203} C_VEL
LIN {X 0,Y 93.376,Z 306.285,A -85,B 0,C 180,E1 -27336.253,E2 -27336.253} C_VEL
LIN {X 0,Y 92.21,Z 309.579,A -85,B 0,C 180,E1 -27337.893,E2 -27337.893} C_VEL
LIN {X 0,Y 91.866,Z 309.713,A -85,B 0,C 180,E1 -27338.69,E2 -27338.69} C_VEL
LIN {X 0,Y 91.796,Z 308.525,A -85,B 0,C 180,E1 -27339.261,E2 -27339.261} C_VEL
LIN {X 0,Y 92.039,Z 305.468,A -85,B 0,C 180,E1 -27339.683,E2 -27339.683} C_VEL
LIN {X 0,Y 91.35,Z 347.756,A -85,B 0,C 180,E1 -27346.937,E2 -27346.937} C_VEL
LIN {X 0,Y 90.88,Z 362.78,A -85,B 0,C 180,E1 -27350.26,E2 -27350.26} C_VEL
LIN {X 0,Y 90.569,Z 376.526,A -85,B 0,C 180,E1 -27354.433,E2 -27354.433} C_VEL
LIN {X 0,Y 90.539,Z 388.134,A -85,B 0,C 180,E1 -27358.887,E2 -27358.887} C_VEL
LIN {X 0,Y 90.793,Z 398.566,A -85,B 0,C 180,E1 -27363.883,E2 -27363.883} C_VEL
LIN {X 0,Y 91.264,Z 407.122,A -85,B 0,C 180,E1 -27368.859,E2 -27368.859} C_VEL
LIN {X 0,Y 92.276,Z 416.347,A -85,B 0,C 180,E1 -27375.459,E2 -27375.459} C_VEL
LIN {X 0,Y 94.717,Z 425.182,A -85,B 0,C 180,E1 -27382.926,E2 -27382.926} C_VEL
LIN {X 0,Y 98.862,Z 432.688,A -85,B 0,C 180,E1 -27389.842,E2 -27389.842} C_VEL
LIN {X 0,Y 105.773,Z 440.063,A -85,B 0,C 180,E1 -27396.726,E2 -27396.726} C_VEL
LIN {X 0,Y 115.158,Z 446.668,A -85,B 0,C 180,E1 -27402.929,E2 -27402.929} C_VEL
LIN {X 0,Y 114.404,Z 446.405,A -85,B 0,C 180,E1 -27403.79,E2 -27403.79} C_VEL
LIN {X 0,Y 105.266,Z 441.53,A -85,B 0,C 180,E1 -27410.63,E2 -27410.63} C_VEL
LIN {X 0,Y 98.344,Z 435.21,A -85,B 0,C 180,E1 -27419.043,E2 -27419.043} C_VEL
LIN {X 0,Y 97.536,Z 434.265,A -85,B 0,C 180,E1 -27420.359,E2 -27420.359} C_VEL
LIN {X 0,Y 92.179,Z 440.933,A -85,B 0,C 180,E1 -27425.202,E2 -27425.202} C_VEL
LIN {X 0,Y 88.125,Z 446.974,A -85,B 0,C 180,E1 -27431.392,E2 -27431.392} C_VEL
LIN {X 0,Y 85.61,Z 451.789,A -85,B 0,C 180,E1 -27438.152,E2 -27438.152} C_VEL
LIN {X 0,Y 84.484,Z 455.484,A -85,B 0,C 180,E1 -27445.223,E2 -27445.223} C_VEL
LIN {X 0,Y 84.354,Z 457.79,A -85,B 0,C 180,E1 -27451.217,E2 -27451.217} C_VEL
LIN {X 0,Y 84.288,Z 459.753,A -85,B 0,C 180,E1 -27459.594,E2 -27459.594} C_VEL
LIN {X 0,Y 86.18,Z 460.533,A -85,B 0,C 180,E1 -27469.033,E2 -27469.033} C_VEL
LIN {X 0,Y 87.916,Z 460.349,A -85,B 0,C 180,E1 -27473.554,E2 -27473.554} C_VEL
LIN {X 0,Y 93.14,Z 458.767,A -85,B 0,C 180,E1 -27481.878,E2 -27481.878} C_VEL
LIN {X 0,Y 96.474,Z 457.403,A -85,B 0,C 180,E1 -27485.641,E2 -27485.641} C_VEL
LIN {X 0,Y 101.694,Z 454.763,A -85,B 0,C 180,E1 -27490.519,E2 -27490.519} C_VEL
LIN {X 0,Y 108.531,Z 450.706,A -85,B 0,C 180,E1 -27495.417,E2 -27495.417} C_VEL
LIN {X 0,Y 115.703,Z 445.749,A -85,B 0,C 180,E1 -27499.394,E2 -27499.394} C_VEL
LIN {X 0,Y 123.419,Z 439.537,A -85,B 0,C 180,E1 -27502.859,E2 -27502.859} C_VEL
LIN {X 0,Y 131.593,Z 431.78,A -85,B 0,C 180,E1 -27505.868,E2 -27505.868} C_VEL
LIN {X 0,Y 138.628,Z 423.896,A -85,B 0,C 180,E1 -27508.115,E2 -27508.115} C_VEL
LIN {X 0,Y 145.878,Z 414.301,A -85,B 0,C 180,E1 -27510.127,E2 -27510.127} C_VEL
LIN {X 0,Y 152.687,Z 403.608,A -85,B 0,C 180,E1 -27511.672,E2 -27511.672} C_VEL
LIN {X 0,Y 158.846,Z 391.463,A -85,B 0,C 180,E1 -27512.915,E2 -27512.915} C_VEL
LIN {X 0,Y 163.466,Z 379.679,A -85,B 0,C 180,E1 -27513.814,E2 -27513.814} C_VEL
LIN {X 0,Y 167.058,Z 367.082,A -85,B 0,C 180,E1 -27514.492,E2 -27514.492} C_VEL
LIN {X 0,Y 169.528,Z 353.357,A -85,B 0,C 180,E1 -27515.004,E2 -27515.004} C_VEL
LIN {X 0,Y 169.746,Z 351.111,A -85,B 0,C 180,E1 -27515.129,E2 -27515.129} C_VEL
LIN {X 0,Y 169.638,Z 350.839,A -85,B 0,C 180,E1 -27515.275,E2 -27515.275} C_VEL
LIN {X 0,Y 168.801,Z 349.05,A -85,B 0,C 180,E1 -27516.415,E2 -27516.415} C_VEL
LIN {X 0,Y 167.37,Z 347.682,A -85,B 0,C 180,E1 -27518.313,E2 -27518.313} C_VEL
LIN {X 0,Y 163.669,Z 346.812,A -85,B 0,C 180,E1 -27524.502,E2 -27524.502} C_VEL
LIN {X 0,Y 163.212,Z 345.926,A -85,B 0,C 180,E1 -27525.885,E2 -27525.885} C_VEL
LIN {X 0,Y 162.831,Z 344.592,A -85,B 0,C 180,E1 -27527.538,E2 -27527.538} C_VEL
LIN {X 0,Y 162.144,Z 343.485,A -85,B 0,C 180,E1 -27532.529,E2 -27532.529} C_VEL
LIN {X 0,Y 162.716,Z 343.937,A -85,B 0,C 180,E1 -27538.144,E2 -27538.144} C_VEL
LIN {X 0,Y 163.03,Z 344.666,A -85,B 0,C 180,E1 -27539.537,E2 -27539.537} C_VEL
LIN {X 0,Y 164.291,Z 348.055,A -85,B 0,C 180,E1 -27543.526,E2 -27543.526} C_VEL
LIN {X 0,Y 165.573,Z 351.515,A -85,B 0,C 180,E1 -27546.551,E2 -27546.551} C_VEL
LIN {X 0,Y 166.941,Z 355.347,A -85,B 0,C 180,E1 -27549.309,E2 -27549.309} C_VEL
LIN {X 0,Y 164.113,Z 367.904,A -85,B 0,C 180,E1 -27549.968,E2 -27549.968} C_VEL
LIN {X 0,Y 160.272,Z 379.619,A -85,B 0,C 180,E1 -27550.763,E2 -27550.763} C_VEL
LIN {X 0,Y 155.294,Z 391.101,A -85,B 0,C 180,E1 -27551.873,E2 -27551.873} C_VEL
LIN {X 0,Y 148.791,Z 402.91,A -85,B 0,C 180,E1 -27553.428,E2 -27553.428} C_VEL
LIN {X 0,Y 141.985,Z 412.833,A -85,B 0,C 180,E1 -27555.169,E2 -27555.169} C_VEL
LIN {X 0,Y 134.37,Z 421.99,A -85,B 0,C 180,E1 -27557.356,E2 -27557.356} C_VEL
LIN {X 0,Y 126.974,Z 429.484,A -85,B 0,C 180,E1 -27559.8,E2 -27559.8} C_VEL
LIN {X 0,Y 118.449,Z 436.785,A -85,B 0,C 180,E1 -27563.133,E2 -27563.133} C_VEL
LIN {X 0,Y 110.384,Z 442.511,A -85,B 0,C 180,E1 -27566.965,E2 -27566.965} C_VEL
LIN {X 0,Y 102.874,Z 446.933,A -85,B 0,C 180,E1 -27571.364,E2 -27571.364} C_VEL
LIN {X 0,Y 96.019,Z 450.198,A -85,B 0,C 180,E1 -27576.385,E2 -27576.385} C_VEL
LIN {X 0,Y 91.898,Z 451.788,A -85,B 0,C 180,E1 -27580.122,E2 -27580.122} C_VEL
LIN {X 0,Y 85.61,Z 453.525,A -85,B 0,C 180,E1 -27587.634,E2 -27587.634} C_VEL
LIN {X 0,Y 82.185,Z 453.89,A -85,B 0,C 180,E1 -27593.237,E2 -27593.237} C_VEL
LIN {X 0,Y 79.952,Z 453.755,A -85,B 0,C 180,E1 -27598.176,E2 -27598.176} C_VEL
LIN {X 0,Y 78.142,Z 453.034,A -85,B 0,C 180,E1 -27604.081,E2 -27604.081} C_VEL
LIN {X 0,Y 76.6,Z 450.739,A -85,B 0,C 180,E1 -27614.029,E2 -27614.029} C_VEL
LIN {X 0,Y 76.865,Z 447.758,A -85,B 0,C 180,E1 -27622.123,E2 -27622.123} C_VEL
LIN {X 0,Y 78.279,Z 443.72,A -85,B 0,C 180,E1 -27630.006,E2 -27630.006} C_VEL
LIN {X 0,Y 81.083,Z 437.52,A -85,B 0,C 180,E1 -27638.73,E2 -27638.73} C_VEL
LIN {X 0,Y 84.608,Z 430.771,A -85,B 0,C 180,E1 -27645.667,E2 -27645.667} C_VEL
LIN {X 0,Y 88.313,Z 423.878,A -85,B 0,C 180,E1 -27650.99,E2 -27650.99} C_VEL
LIN {X 0,Y 92.721,Z 415.55,A -85,B 0,C 180,E1 -27655.843,E2 -27655.843} C_VEL
LIN {X 0,Y 97.676,Z 405.265,A -85,B 0,C 180,E1 -27660.248,E2 -27660.248} C_VEL
LIN {X 0,Y 101.942,Z 395.121,A -85,B 0,C 180,E1 -27663.477,E2 -27663.477} C_VEL
LIN {X 0,Y 105.911,Z 384.033,A -85,B 0,C 180,E1 -27666.086,E2 -27666.086} C_VEL
LIN {X 0,Y 108.847,Z 372.916,A -85,B 0,C 180,E1 -27668.133,E2 -27668.133} C_VEL
LIN {X 0,Y 111.72,Z 359.869,A -85,B 0,C 180,E1 -27669.633,E2 -27669.633} C_VEL
LIN {X 0,Y 113.527,Z 346.426,A -85,B 0,C 180,E1 -27670.642,E2 -27670.642} C_VEL
LIN {X 0,Y 116.321,Z 312.926,A -85,B 0,C 180,E1 -27672.228,E2 -27672.228} C_VEL
LIN {X 0,Y 111.616,Z 302.496,A -85,B 0,C 180,E1 -27676.319,E2 -27676.319} C_VEL
LIN {X 0,Y 107.584,Z 295.213,A -85,B 0,C 180,E1 -27680.298,E2 -27680.298} C_VEL
LIN {X 0,Y 104.069,Z 289.554,A -85,B 0,C 180,E1 -27684.366,E2 -27684.366} C_VEL
LIN {X 0,Y 102.636,Z 287.368,A -85,B 0,C 180,E1 -27686.244,E2 -27686.244} C_VEL
LIN {X 0,Y 100.419,Z 290.416,A -85,B 0,C 180,E1 -27688.392,E2 -27688.392} C_VEL
LIN {X 0,Y 96.865,Z 303.367,A -85,B 0,C 180,E1 -27690.849,E2 -27690.849} C_VEL
LIN {X 0,Y 94.499,Z 310.903,A -85,B 0,C 180,E1 -27693.004,E2 -27693.004} C_VEL
LIN {X 0,Y 92.909,Z 314.826,A -85,B 0,C 180,E1 -27694.952,E2 -27694.952} C_VEL
LIN {X 0,Y 91.755,Z 316.589,A -85,B 0,C 180,E1 -27696.861,E2 -27696.861} C_VEL
LIN {X 0,Y 87.64,Z 336.381,A -85,B 0,C 180,E1 -27700.986,E2 -27700.986} C_VEL
LIN {X 0,Y 85.365,Z 347.293,A -85,B 0,C 180,E1 -27704.326,E2 -27704.326} C_VEL
LIN {X 0,Y 84.615,Z 350.444,A -85,B 0,C 180,E1 -27705.877,E2 -27705.877} C_VEL
LIN {X 0,Y 84.3,Z 351.521,A -85,B 0,C 180,E1 -27706.745,E2 -27706.745} C_VEL
LIN {X 0,Y 84.167,Z 351.351,A -85,B 0,C 180,E1 -27707.95,E2 -27707.95} C_VEL
LIN {X 0,Y 84.468,Z 349.032,A -85,B 0,C 180,E1 -27708.45,E2 -27708.45} C_VEL
LIN {X 0,Y 84.751,Z 347.293,A -85,B 0,C 180,E1 -27708.64,E2 -27708.64} C_VEL
LIN {X 0,Y 84.469,Z 361.206,A -85,B 0,C 180,E1 -27711.928,E2 -27711.928} C_VEL
LIN {X 0,Y 84.269,Z 373.769,A -85,B 0,C 180,E1 -27715.874,E2 -27715.874} C_VEL
LIN {X 0,Y 84.424,Z 385.57,A -85,B 0,C 180,E1 -27720.595,E2 -27720.595} C_VEL
LIN {X 0,Y 84.819,Z 395.366,A -85,B 0,C 180,E1 -27725.408,E2 -27725.408} C_VEL
LIN {X 0,Y 85.446,Z 404.128,A -85,B 0,C 180,E1 -27730.664,E2 -27730.664} C_VEL
LIN {X 0,Y 86.412,Z 412.182,A -85,B 0,C 180,E1 -27736.537,E2 -27736.537} C_VEL
LIN {X 0,Y 88.567,Z 420.341,A -85,B 0,C 180,E1 -27743.375,E2 -27743.375} C_VEL
LIN {X 0,Y 93.362,Z 429.485,A -85,B 0,C 180,E1 -27751.798,E2 -27751.798} C_VEL
LIN {X 0,Y 100.577,Z 437.331,A -85,B 0,C 180,E1 -27758.968,E2 -27758.968} C_VEL
LIN {X 0,Y 104.857,Z 440.773,A -85,B 0,C 180,E1 -27762.085,E2 -27762.085} C_VEL
LIN {X 0,Y 106.57,Z 442.064,A -85,B 0,C 180,E1 -27763.491,E2 -27763.491} C_VEL
LIN {X 0,Y 98.611,Z 437.071,A -85,B 0,C 180,E1 -27770.096,E2 -27770.096} C_VEL
LIN {X 0,Y 92.946,Z 431.676,A -85,B 0,C 180,E1 -27777.236,E2 -27777.236} C_VEL
LIN {X 0,Y 88.79,Z 436.452,A -85,B 0,C 180,E1 -27780.27,E2 -27780.27} C_VEL
LIN {X 0,Y 84.172,Z 442.298,A -85,B 0,C 180,E1 -27785.319,E2 -27785.319} C_VEL
LIN {X 0,Y 80.36,Z 448.035,A -85,B 0,C 180,E1 -27792.17,E2 -27792.17} C_VEL
LIN {X 0,Y 78.137,Z 452.56,A -85,B 0,C 180,E1 -27799.631,E2 -27799.631} C_VEL
LIN {X 0,Y 77.323,Z 456.47,A -85,B 0,C 180,E1 -27808.821,E2 -27808.821} C_VEL
LIN {X 0,Y 77.316,Z 457.163,A -85,B 0,C 180,E1 -27810.901,E2 -27810.901} C_VEL
LIN {X 0,Y 77.284,Z 459.348,A -85,B 0,C 180,E1 -27820.473,E2 -27820.473} C_VEL
LIN {X 0,Y 79.483,Z 460.2,A -85,B 0,C 180,E1 -27830.707,E2 -27830.707} C_VEL
LIN {X 0,Y 81.425,Z 460.061,A -85,B 0,C 180,E1 -27835.561,E2 -27835.561} C_VEL
LIN {X 0,Y 84.059,Z 459.524,A -85,B 0,C 180,E1 -27840.103,E2 -27840.103} C_VEL
LIN {X 0,Y 90.787,Z 457.251,A -85,B 0,C 180,E1 -27848.258,E2 -27848.258} C_VEL
LIN {X 0,Y 95.772,Z 454.995,A -85,B 0,C 180,E1 -27852.793,E2 -27852.793} C_VEL
LIN {X 0,Y 103.662,Z 450.712,A -85,B 0,C 180,E1 -27858.219,E2 -27858.219} C_VEL
LIN {X 0,Y 111.221,Z 445.843,A -85,B 0,C 180,E1 -27862.166,E2 -27862.166} C_VEL
LIN {X 0,Y 119.276,Z 439.727,A -85,B 0,C 180,E1 -27865.572,E2 -27865.572} C_VEL
LIN {X 0,Y 127.758,Z 432.134,A -85,B 0,C 180,E1 -27868.495,E2 -27868.495} C_VEL
LIN {X 0,Y 136.497,Z 422.633,A -85,B 0,C 180,E1 -27871.073,E2 -27871.073} C_VEL
LIN {X 0,Y 144.03,Z 412.844,A -85,B 0,C 180,E1 -27872.931,E2 -27872.931} C_VEL
LIN {X 0,Y 151.034,Z 401.785,A -85,B 0,C 180,E1 -27874.358,E2 -27874.358} C_VEL
LIN {X 0,Y 156.551,Z 391.002,A -85,B 0,C 180,E1 -27875.371,E2 -27875.371} C_VEL
LIN {X 0,Y 161.287,Z 379.161,A -85,B 0,C 180,E1 -27876.208,E2 -27876.208} C_VEL
LIN {X 0,Y 164.957,Z 366.46,A -85,B 0,C 180,E1 -27876.841,E2 -27876.841} C_VEL
LIN {X 0,Y 167.072,Z 355.243,A -85,B 0,C 180,E1 -27877.286,E2 -27877.286} C_VEL
LIN {X 0,Y 165.154,Z 350.303,A -85,B 0,C 180,E1 -27880.906,E2 -27880.906} C_VEL
LIN {X 0,Y 163.963,Z 347.577,A -85,B 0,C 180,E1 -27883.663,E2 -27883.663} C_VEL
LIN {X 0,Y 163.212,Z 345.926,A -85,B 0,C 180,E1 -27885.885,E2 -27885.885} C_VEL
LIN {X 0,Y 162.843,Z 345.236,A -85,B 0,C 180,E1 -27887.228,E2 -27887.228} C_VEL
LIN {X 0,Y 162.277,Z 345.588,A -85,B 0,C 180,E1 -27889.294,E2 -27889.294} C_VEL
LIN {X 0,Y 161.548,Z 348.161,A -85,B 0,C 180,E1 -27892.731,E2 -27892.731} C_VEL
LIN {X 0,Y 161.385,Z 350.261,A -85,B 0,C 180,E1 -27895.54,E2 -27895.54} C_VEL
LIN {X 0,Y 161.527,Z 350.755,A -85,B 0,C 180,E1 -27896.975,E2 -27896.975} C_VEL
LIN {X 0,Y 161.859,Z 351.342,A -85,B 0,C 180,E1 -27898.792,E2 -27898.792} C_VEL
LIN {X 0,Y 162.85,Z 354.838,A -85,B 0,C 180,E1 -27902.938,E2 -27902.938} C_VEL
LIN {X 0,Y 164.009,Z 358.799,A -85,B 0,C 180,E1 -27906.413,E2 -27906.413} C_VEL
LIN {X 0,Y 164.271,Z 359.701,A -85,B 0,C 180,E1 -27907.125,E2 -27907.125} C_VEL
LIN {X 0,Y 160.866,Z 372.431,A -85,B 0,C 180,E1 -27907.827,E2 -27907.827} C_VEL
LIN {X 0,Y 156.402,Z 384.351,A -85,B 0,C 180,E1 -27908.688,E2 -27908.688} C_VEL
LIN {X 0,Y 150.702,Z 396.011,A -85,B 0,C 180,E1 -27909.9,E2 -27909.9} C_VEL
LIN {X 0,Y 143.437,Z 407.683,A -85,B 0,C 180,E1 -27911.513,E2 -27911.513} C_VEL
LIN {X 0,Y 137.069,Z 416.054,A -85,B 0,C 180,E1 -27913.06,E2 -27913.06} C_VEL
LIN {X 0,Y 129.351,Z 424.585,A -85,B 0,C 180,E1 -27915.157,E2 -27915.157} C_VEL
LIN {X 0,Y 120.174,Z 432.998,A -85,B 0,C 180,E1 -27918.146,E2 -27918.146} C_VEL
LIN {X 0,Y 112.841,Z 438.608,A -85,B 0,C 180,E1 -27920.906,E2 -27920.906} C_VEL
LIN {X 0,Y 104.496,Z 444.021,A -85,B 0,C 180,E1 -27924.786,E2 -27924.786} C_VEL
LIN {X 0,Y 96.668,Z 448.163,A -85,B 0,C 180,E1 -27929.267,E2 -27929.267} C_VEL
LIN {X 0,Y 91.828,Z 450.28,A -85,B 0,C 180,E1 -27932.671,E2 -27932.671} C_VEL
LIN {X 0,Y 87.295,Z 451.917,A -85,B 0,C 180,E1 -27936.39,E2 -27936.39} C_VEL
LIN {X 0,Y 83.201,Z 453.128,A -85,B 0,C 180,E1 -27940.524,E2 -27940.524} C_VEL
LIN {X 0,Y 79.571,Z 453.878,A -85,B 0,C 180,E1 -27945.05,E2 -27945.05} C_VEL
LIN {X 0,Y 76.379,Z 454.195,A -85,B 0,C 180,E1 -27949.91,E2 -27949.91} C_VEL
LIN {X 0,Y 73.768,Z 454.107,A -85,B 0,C 180,E1 -27955.144,E2 -27955.144} C_VEL
LIN {X 0,Y 71.341,Z 453.324,A -85,B 0,C 180,E1 -27962.455,E2 -27962.455} C_VEL
LIN {X 0,Y 69.596,Z 451.258,A -85,B 0,C 180,E1 -27972.372,E2 -27972.372} C_VEL
LIN {X 0,Y 69.676,Z 448.364,A -85,B 0,C 180,E1 -27981.304,E2 -27981.304} C_VEL
LIN {X 0,Y 71.062,Z 444.422,A -85,B 0,C 180,E1 -27990.006,E2 -27990.006} C_VEL
LIN {X 0,Y 73.52,Z 439.35,A -85,B 0,C 180,E1 -27998.25,E2 -27998.25} C_VEL
LIN {X 0,Y 77.027,Z 432.958,A -85,B 0,C 180,E1 -28005.892,E2 -28005.892} C_VEL
LIN {X 0,Y 81.703,Z 424.966,A -85,B 0,C 180,E1 -28012.779,E2 -28012.779} C_VEL
LIN {X 0,Y 86.37,Z 416.792,A -85,B 0,C 180,E1 -28017.902,E2 -28017.902} C_VEL
LIN {X 0,Y 91.574,Z 406.793,A -85,B 0,C 180,E1 -28022.501,E2 -28022.501} C_VEL
LIN {X 0,Y 96.676,Z 395.499,A -85,B 0,C 180,E1 -28026.209,E2 -28026.209} C_VEL
LIN {X 0,Y 100.863,Z 384.426,A -85,B 0,C 180,E1 -28028.843,E2 -28028.843} C_VEL
LIN {X 0,Y 103.98,Z 373.342,A -85,B 0,C 180,E1 -28030.908,E2 -28030.908} C_VEL
LIN {X 0,Y 107.025,Z 360.139,A -85,B 0,C 180,E1 -28032.417,E2 -28032.417} C_VEL
LIN {X 0,Y 108.845,Z 347.466,A -85,B 0,C 180,E1 -28033.372,E2 -28033.372} C_VEL
LIN {X 0,Y 111.675,Z 315.511,A -85,B 0,C 180,E1 -28034.884,E2 -28034.884} C_VEL
LIN {X 0,Y 108.119,Z 307.263,A -85,B 0,C 180,E1 -28038.391,E2 -28038.391} C_VEL
LIN {X 0,Y 104.222,Z 299.777,A -85,B 0,C 180,E1 -28042.757,E2 -28042.757} C_VEL
LIN {X 0,Y 102.268,Z 296.372,A -85,B 0,C 180,E1 -28045.26,E2 -28045.26} C_VEL
LIN {X 0,Y 102.062,Z 296.383,A -85,B 0,C 180,E1 -28045.483,E2 -28045.483} C_VEL
LIN {X 0,Y 98.451,Z 308.325,A -85,B 0,C 180,E1 -28047.77,E2 -28047.77} C_VEL
LIN {X 0,Y 95.822,Z 315.751,A -85,B 0,C 180,E1 -28049.937,E2 -28049.937} C_VEL
LIN {X 0,Y 93.774,Z 320.201,A -85,B 0,C 180,E1 -28052.154,E2 -28052.154} C_VEL
LIN {X 0,Y 92.797,Z 321.935,A -85,B 0,C 180,E1 -28053.427,E2 -28053.427} C_VEL
LIN {X 0,Y 88.826,Z 339.25,A -85,B 0,C 180,E1 -28056.849,E2 -28056.849} C_VEL
LIN {X 0,Y 86.235,Z 349.825,A -85,B 0,C 180,E1 -28059.889,E2 -28059.889} C_VEL
LIN {X 0,Y 84.825,Z 354.568,A -85,B 0,C 180,E1 -28061.897,E2 -28061.897} C_VEL
LIN {X 0,Y 83.724,Z 357.363,A -85,B 0,C 180,E1 -28064.011,E2 -28064.011} C_VEL
LIN {X 0,Y 83.107,Z 358.447,A -85,B 0,C 180,E1 -28066.084,E2 -28066.084} C_VEL
LIN {X 0,Y 80.426,Z 367.51,A -85,B 0,C 180,E1 -28069.297,E2 -28069.297} C_VEL
LIN {X 0,Y 78.578,Z 372.999,A -85,B 0,C 180,E1 -28072.291,E2 -28072.291} C_VEL
LIN {X 0,Y 77.598,Z 375.978,A -85,B 0,C 180,E1 -28074.802,E2 -28074.802} C_VEL
LIN {X 0,Y 77.349,Z 377.578,A -85,B 0,C 180,E1 -28078.305,E2 -28078.305} C_VEL
LIN {X 0,Y 78.222,Z 375.711,A -85,B 0,C 180,E1 -28079.478,E2 -28079.478} C_VEL
LIN {X 0,Y 78.71,Z 388.041,A -85,B 0,C 180,E1 -28085.122,E2 -28085.122} C_VEL
LIN {X 0,Y 79.393,Z 397.033,A -85,B 0,C 180,E1 -28090.196,E2 -28090.196} C_VEL
LIN {X 0,Y 80.341,Z 405.163,A -85,B 0,C 180,E1 -28095.774,E2 -28095.774} C_VEL
LIN {X 0,Y 82.59,Z 415.007,A -85,B 0,C 180,E1 -28103.84,E2 -28103.84} C_VEL
LIN {X 0,Y 87.284,Z 424.841,A -85,B 0,C 180,E1 -28112.921,E2 -28112.921} C_VEL
LIN {X 0,Y 93.56,Z 432.349,A -85,B 0,C 180,E1 -28119.679,E2 -28119.679} C_VEL
LIN {X 0,Y 97.113,Z 435.608,A -85,B 0,C 180,E1 -28122.567,E2 -28122.567} C_VEL
LIN {X 0,Y 97.89,Z 436.385,A -85,B 0,C 180,E1 -28124.108,E2 -28124.108} C_VEL
LIN {X 0,Y 89.627,Z 429.625,A -85,B 0,C 180,E1 -28132.704,E2 -28132.704} C_VEL
LIN {X 0,Y 88.828,Z 428.871,A -85,B 0,C 180,E1 -28133.766,E2 -28133.766} C_VEL
LIN {X 0,Y 83.882,Z 434.239,A -85,B 0,C 180,E1 -28136.912,E2 -28136.912} C_VEL
LIN {X 0,Y 77.826,Z 441.492,A -85,B 0,C 180,E1 -28143.152,E2 -28143.152} C_VEL
LIN {X 0,Y 73.68,Z 447.322,A -85,B 0,C 180,E1 -28150.491,E2 -28150.491} C_VEL
LIN {X 0,Y 71.192,Z 451.932,A -85,B 0,C 180,E1 -28158.607,E2 -28158.607} C_VEL
LIN {X 0,Y 70.382,Z 454.382,A -85,B 0,C 180,E1 -28164.263,E2 -28164.263} C_VEL
LIN {X 0,Y 70.28,Z 456.441,A -85,B 0,C 180,E1 -28170.287,E2 -28170.287} C_VEL
LIN {X 0,Y 70.294,Z 458.937,A -85,B 0,C 180,E1 -28181.528,E2 -28181.528} C_VEL
LIN {X 0,Y 72.852,Z 459.866,A -85,B 0,C 180,E1 -28192.692,E2 -28192.692} C_VEL
LIN {X 0,Y 75.056,Z 459.763,A -85,B 0,C 180,E1 -28197.91,E2 -28197.91} C_VEL
LIN {X 0,Y 77.978,Z 459.289,A -85,B 0,C 180,E1 -28202.729,E2 -28202.729} C_VEL
LIN {X 0,Y 85.299,Z 457.099,A -85,B 0,C 180,E1 -28211.227,E2 -28211.227} C_VEL
LIN {X 0,Y 90.132,Z 455.165,A -85,B 0,C 180,E1 -28215.432,E2 -28215.432} C_VEL
LIN {X 0,Y 99.062,Z 450.718,A -85,B 0,C 180,E1 -28221.29,E2 -28221.29} C_VEL
LIN {X 0,Y 107.022,Z 445.936,A -85,B 0,C 180,E1 -28225.163,E2 -28225.163} C_VEL
LIN {X 0,Y 116.863,Z 438.805,A -85,B 0,C 180,E1 -28228.971,E2 -28228.971} C_VEL
LIN {X 0,Y 125.71,Z 431.022,A -85,B 0,C 180,E1 -28231.698,E2 -28231.698} C_VEL
LIN {X 0,Y 133.22,Z 423.12,A -85,B 0,C 180,E1 -28233.736,E2 -28233.736} C_VEL
LIN {X 0,Y 140.954,Z 413.499,A -85,B 0,C 180,E1 -28235.49,E2 -28235.49} C_VEL
LIN {X 0,Y 148.122,Z 402.765,A -85,B 0,C 180,E1 -28236.815,E2 -28236.815} C_VEL
LIN {X 0,Y 154.555,Z 390.585,A -85,B 0,C 180,E1 -28237.888,E2 -28237.888} C_VEL
LIN {X 0,Y 159.659,Z 377.95,A -85,B 0,C 180,E1 -28238.698,E2 -28238.698} C_VEL
LIN {X 0,Y 163.284,Z 365.369,A -85,B 0,C 180,E1 -28239.26,E2 -28239.26} C_VEL
LIN {X 0,Y 164.465,Z 359.543,A -85,B 0,C 180,E1 -28239.542,E2 -28239.542} C_VEL
LIN {X 0,Y 163.141,Z 355.549,A -85,B 0,C 180,E1 -28242.934,E2 -28242.934} C_VEL
LIN {X 0,Y 162.114,Z 352.922,A -85,B 0,C 180,E1 -28246.206,E2 -28246.206} C_VEL
LIN {X 0,Y 161.758,Z 351.492,A -85,B 0,C 180,E1 -28248.09,E2 -28248.09} C_VEL
LIN {X 0,Y 161.224,Z 350.536,A -85,B 0,C 180,E1 -28252.486,E2 -28252.486} C_VEL
LIN {X 0,Y 161.527,Z 350.755,A -85,B 0,C 180,E1 -28256.975,E2 -28256.975} C_VEL
LIN {X 0,Y 161.638,Z 351.585,A -85,B 0,C 180,E1 -28258.088,E2 -28258.088} C_VEL
LIN {X 0,Y 161.591,Z 354.194,A -85,B 0,C 180,E1 -28259.456,E2 -28259.456} C_VEL
LIN {X 0,Y 161.139,Z 360.671,A -85,B 0,C 180,E1 -28261.993,E2 -28261.993} C_VEL
LIN {X 0,Y 161.255,Z 362.485,A -85,B 0,C 180,E1 -28263.29,E2 -28263.29} C_VEL
LIN {X 0,Y 161.631,Z 364.305,A -85,B 0,C 180,E1 -28264.882,E2 -28264.882} C_VEL
LIN {X 0,Y 157.651,Z 377.077,A -85,B 0,C 180,E1 -28265.612,E2 -28265.612} C_VEL
LIN {X 0,Y 152.942,Z 388.246,A -85,B 0,C 180,E1 -28266.455,E2 -28266.455} C_VEL
LIN {X 0,Y 147.12,Z 399.181,A -85,B 0,C 180,E1 -28267.619,E2 -28267.619} C_VEL
LIN {X 0,Y 140.503,Z 409.118,A -85,B 0,C 180,E1 -28268.944,E2 -28268.944} C_VEL
LIN {X 0,Y 132.349,Z 419.111,A -85,B 0,C 180,E1 -28270.789,E2 -28270.789} C_VEL
LIN {X 0,Y 124.181,Z 427.387,A -85,B 0,C 180,E1 -28272.898,E2 -28272.898} C_VEL
LIN {X 0,Y 114.997,Z 435.107,A -85,B 0,C 180,E1 -28275.744,E2 -28275.744} C_VEL
LIN {X 0,Y 107.14,Z 440.59,A -85,B 0,C 180,E1 -28278.596,E2 -28278.596} C_VEL
LIN {X 0,Y 98.766,Z 445.465,A -85,B 0,C 180,E1 -28282.336,E2 -28282.336} C_VEL
LIN {X 0,Y 90.609,Z 449.305,A -85,B 0,C 180,E1 -28286.888,E2 -28286.888} C_VEL
LIN {X 0,Y 83.12,Z 452.044,A -85,B 0,C 180,E1 -28292.282,E2 -28292.282} C_VEL
LIN {X 0,Y 78.58,Z 453.301,A -85,B 0,C 180,E1 -28296.406,E2 -28296.406} C_VEL
LIN {X 0,Y 73.931,Z 454.205,A -85,B 0,C 180,E1 -28301.717,E2 -28301.717} C_VEL
LIN {X 0,Y 67.848,Z 454.454,A -85,B 0,C 180,E1 -28311.582,E2 -28311.582} C_VEL
LIN {X 0,Y 64.627,Z 453.618,A -85,B 0,C 180,E1 -28320.459,E2 -28320.459} C_VEL
LIN {X 0,Y 62.674,Z 451.776,A -85,B 0,C 180,E1 -28330.349,E2 -28330.349} C_VEL
LIN {X 0,Y 62.476,Z 448.971,A -85,B 0,C 180,E1 -28340.293,E2 -28340.293} C_VEL
LIN {X 0,Y 63.852,Z 445.117,A -85,B 0,C 180,E1 -28350.007,E2 -28350.007} C_VEL
LIN {X 0,Y 66.426,Z 440.144,A -85,B 0,C 180,E1 -28359.138,E2 -28359.138} C_VEL
LIN {X 0,Y 70.185,Z 433.903,A -85,B 0,C 180,E1 -28367.489,E2 -28367.489} C_VEL
LIN {X 0,Y 75.187,Z 426.053,A -85,B 0,C 180,E1 -28374.881,E2 -28374.881} C_VEL
LIN {X 0,Y 80.146,Z 418.031,A -85,B 0,C 180,E1 -28380.286,E2 -28380.286} C_VEL
LIN {X 0,Y 85.636,Z 408.267,A -85,B 0,C 180,E1 -28385.069,E2 -28385.069} C_VEL
LIN {X 0,Y 91.038,Z 397.273,A -85,B 0,C 180,E1 -28388.853,E2 -28388.853} C_VEL
LIN {X 0,Y 95.422,Z 386.543,A -85,B 0,C 180,E1 -28391.525,E2 -28391.525} C_VEL
LIN {X 0,Y 99.049,Z 374.893,A -85,B 0,C 180,E1 -28393.779,E2 -28393.779} C_VEL
LIN {X 0,Y 102.302,Z 361.937,A -85,B 0,C 180,E1 -28395.309,E2 -28395.309} C_VEL
LIN {X 0,Y 104.384,Z 348.787,A -85,B 0,C 180,E1 -28396.326,E2 -28396.326} C_VEL
LIN {X 0,Y 107.27,Z 318.149,A -85,B 0,C 180,E1 -28397.772,E2 -28397.772} C_VEL
LIN {X 0,Y 104.484,Z 311.43,A -85,B 0,C 180,E1 -28400.936,E2 -28400.936} C_VEL
LIN {X 0,Y 102.445,Z 307.196,A -85,B 0,C 180,E1 -28403.471,E2 -28403.471} C_VEL
LIN {X 0,Y 98.878,Z 317.062,A -85,B 0,C 180,E1 -28405.807,E2 -28405.807} C_VEL
LIN {X 0,Y 96.344,Z 322.847,A -85,B 0,C 180,E1 -28407.916,E2 -28407.916} C_VEL
LIN {X 0,Y 94.466,Z 326.216,A -85,B 0,C 180,E1 -28409.854,E2 -28409.854} C_VEL
LIN {X 0,Y 90.335,Z 342.587,A -85,B 0,C 180,E1 -28412.957,E2 -28412.957} C_VEL
LIN {X 0,Y 87.189,Z 353.484,A -85,B 0,C 180,E1 -28415.915,E2 -28415.915} C_VEL
LIN {X 0,Y 85.295,Z 358.528,A -85,B 0,C 180,E1 -28417.917,E2 -28417.917} C_VEL
LIN {X 0,Y 83.294,Z 362.73,A -85,B 0,C 180,E1 -28420.755,E2 -28420.755} C_VEL
LIN {X 0,Y 82.432,Z 364.237,A -85,B 0,C 180,E1 -28422.479,E2 -28422.479} C_VEL
LIN {X 0,Y 79.533,Z 371.869,A -85,B 0,C 180,E1 -28425.281,E2 -28425.281} C_VEL
LIN {X 0,Y 77.262,Z 377.142,A -85,B 0,C 180,E1 -28428.189,E2 -28428.189} C_VEL
LIN {X 0,Y 75.745,Z 380.539,A -85,B 0,C 180,E1 -28430.89,E2 -28430.89} C_VEL
LIN {X 0,Y 75.197,Z 381.839,A -85,B 0,C 180,E1 -28432.413,E2 -28432.413} C_VEL
LIN {X 0,Y 74.386,Z 384.563,A -85,B 0,C 180,E1 -28438.238,E2 -28438.238} C_VEL
LIN {X 0,Y 73.041,Z 388.538,A -85,B 0,C 180,E1 -28441.377,E2 -28441.377} C_VEL
LIN {X 0,Y 72.117,Z 392.396,A -85,B 0,C 180,E1 -28445.591,E2 -28445.591} C_VEL
LIN {X 0,Y 72.014,Z 393.794,A -85,B 0,C 180,E1 -28447.71,E2 -28447.71} C_VEL
LIN {X 0,Y 72.564,Z 395.197,A -85,B 0,C 180,E1 -28451.168,E2 -28451.168} C_VEL
LIN {X 0,Y 73.305,Z 394.957,A -85,B 0,C 180,E1 -28452.456,E2 -28452.456} C_VEL
LIN {X 0,Y 73.911,Z 394.296,A -85,B 0,C 180,E1 -28452.876,E2 -28452.876} C_VEL
LIN {X 0,Y 74.954,Z 401.131,A -85,B 0,C 180,E1 -28457.741,E2 -28457.741} C_VEL
LIN {X 0,Y 77.225,Z 410.489,A -85,B 0,C 180,E1 -28465.467,E2 -28465.467} C_VEL
LIN {X 0,Y 82.231,Z 420.964,A -85,B 0,C 180,E1 -28475.231,E2 -28475.231} C_VEL
LIN {X 0,Y 88.806,Z 428.901,A -85,B 0,C 180,E1 -28482.273,E2 -28482.273} C_VEL
LIN {X 0,Y 90.016,Z 430.224,A -85,B 0,C 180,E1 -28484.641,E2 -28484.641} C_VEL
LIN {X 0,Y 85.129,Z 425.968,A -85,B 0,C 180,E1 -28490.044,E2 -28490.044} C_VEL
LIN {X 0,Y 79.249,Z 431.988,A -85,B 0,C 180,E1 -28493.188,E2 -28493.188} C_VEL
LIN {X 0,Y 72.565,Z 439.599,A -85,B 0,C 180,E1 -28499.431,E2 -28499.431} C_VEL
LIN {X 0,Y 68.392,Z 444.795,A -85,B 0,C 180,E1 -28505.723,E2 -28505.723} C_VEL
LIN {X 0,Y 64.994,Z 449.888,A -85,B 0,C 180,E1 -28514.309,E2 -28514.309} C_VEL
LIN {X 0,Y 63.335,Z 453.824,A -85,B 0,C 180,E1 -28523.622,E2 -28523.622} C_VEL
LIN {X 0,Y 63.211,Z 455.839,A -85,B 0,C 180,E1 -28529.993,E2 -28529.993} C_VEL
LIN {X 0,Y 62.924,Z 457.369,A -85,B 0,C 180,E1 -28536.406,E2 -28536.406} C_VEL
LIN {X 0,Y 63.345,Z 458.502,A -85,B 0,C 180,E1 -28542.813,E2 -28542.813} C_VEL
LIN {X 0,Y 64.463,Z 459.222,A -85,B 0,C 180,E1 -28549.084,E2 -28549.084} C_VEL
LIN {X 0,Y 68.841,Z 459.466,A -85,B 0,C 180,E1 -28560.686,E2 -28560.686} C_VEL
LIN {X 0,Y 75.826,Z 458.201,A -85,B 0,C 180,E1 -28570.443,E2 -28570.443} C_VEL
LIN {X 0,Y 84.621,Z 455.302,A -85,B 0,C 180,E1 -28578.363,E2 -28578.363} C_VEL
LIN {X 0,Y 92.132,Z 452.032,A -85,B 0,C 180,E1 -28583.213,E2 -28583.213} C_VEL
LIN {X 0,Y 100.279,Z 447.717,A -85,B 0,C 180,E1 -28587.239,E2 -28587.239} C_VEL
LIN {X 0,Y 110.396,Z 441.219,A -85,B 0,C 180,E1 -28591.078,E2 -28591.078} C_VEL
LIN {X 0,Y 119.431,Z 434.106,A -85,B 0,C 180,E1 -28593.809,E2 -28593.809} C_VEL
LIN {X 0,Y 127.163,Z 426.903,A -85,B 0,C 180,E1 -28595.762,E2 -28595.762} C_VEL
LIN {X 0,Y 134.989,Z 418.206,A -85,B 0,C 180,E1 -28597.528,E2 -28597.528} C_VEL
LIN {X 0,Y 142.232,Z 408.658,A -85,B 0,C 180,E1 -28598.843,E2 -28598.843} C_VEL
LIN {X 0,Y 148.765,Z 398.22,A -85,B 0,C 180,E1 -28599.865,E2 -28599.865} C_VEL
LIN {X 0,Y 154.507,Z 386.602,A -85,B 0,C 180,E1 -28600.699,E2 -28600.699} C_VEL
LIN {X 0,Y 159.197,Z 374.112,A -85,B 0,C 180,E1 -28601.373,E2 -28601.373} C_VEL
LIN {X 0,Y 161.925,Z 364.175,A -85,B 0,C 180,E1 -28601.766,E2 -28601.766} C_VEL
LIN {X 0,Y 161.106,Z 361.083,A -85,B 0,C 180,E1 -28604.827,E2 -28604.827} C_VEL
LIN {X 0,Y 160.389,Z 358.366,A -85,B 0,C 180,E1 -28608.628,E2 -28608.628} C_VEL
LIN {X 0,Y 159.991,Z 357.546,A -85,B 0,C 180,E1 -28612.428,E2 -28612.428} C_VEL
LIN {X 0,Y 160.432,Z 357.963,A -85,B 0,C 180,E1 -28618.049,E2 -28618.049} C_VEL
LIN {X 0,Y 161.035,Z 361.366,A -85,B 0,C 180,E1 -28622.189,E2 -28622.189} C_VEL
LIN {X 0,Y 161.255,Z 362.485,A -85,B 0,C 180,E1 -28623.29,E2 -28623.29} C_VEL
LIN {X 0,Y 161.227,Z 363.682,A -85,B 0,C 180,E1 -28623.842,E2 -28623.842} C_VEL
LIN {X 0,Y 160.705,Z 366.118,A -85,B 0,C 180,E1 -28624.186,E2 -28624.186} C_VEL
LIN {X 0,Y 159.497,Z 369.992,A -85,B 0,C 180,E1 -28624.173,E2 -28624.173} C_VEL
LIN {X 0,Y 155.39,Z 379.737,A -85,B 0,C 180,E1 -28623.353,E2 -28623.353} C_VEL
LIN {X 0,Y 154.155,Z 382.563,A -85,B 0,C 180,E1 -28623.408,E2 -28623.408} C_VEL
LIN {X 0,Y 148.875,Z 393.522,A -85,B 0,C 180,E1 -28624.287,E2 -28624.287} C_VEL
LIN {X 0,Y 142.085,Z 404.714,A -85,B 0,C 180,E1 -28625.505,E2 -28625.505} C_VEL
LIN {X 0,Y 134.509,Z 414.68,A -85,B 0,C 180,E1 -28626.939,E2 -28626.939} C_VEL
LIN {X 0,Y 126.2,Z 423.68,A -85,B 0,C 180,E1 -28628.729,E2 -28628.729} C_VEL
LIN {X 0,Y 117.736,Z 431.292,A -85,B 0,C 180,E1 -28630.844,E2 -28630.844} C_VEL
LIN {X 0,Y 108.45,Z 438.194,A -85,B 0,C 180,E1 -28633.594,E2 -28633.594} C_VEL
LIN {X 0,Y 98.76,Z 444.047,A -85,B 0,C 180,E1 -28637.155,E2 -28637.155} C_VEL
LIN {X 0,Y 90.355,Z 448.152,A -85,B 0,C 180,E1 -28641.046,E2 -28641.046} C_VEL
LIN {X 0,Y 83.708,Z 450.788,A -85,B 0,C 180,E1 -28644.823,E2 -28644.823} C_VEL
LIN {X 0,Y 74.412,Z 453.478,A -85,B 0,C 180,E1 -28651.798,E2 -28651.798} C_VEL
LIN {X 0,Y 68.428,Z 454.548,A -85,B 0,C 180,E1 -28658.044,E2 -28658.044} C_VEL
LIN {X 0,Y 62.218,Z 454.803,A -85,B 0,C 180,E1 -28667.342,E2 -28667.342} C_VEL
LIN {X 0,Y 57.97,Z 453.904,A -85,B 0,C 180,E1 -28678.068,E2 -28678.068} C_VEL
LIN {X 0,Y 55.832,Z 452.295,A -85,B 0,C 180,E1 -28687.821,E2 -28687.821} C_VEL
LIN {X 0,Y 55.305,Z 449.578,A -85,B 0,C 180,E1 -28699.02,E2 -28699.02} C_VEL
LIN {X 0,Y 56.618,Z 445.815,A -85,B 0,C 180,E1 -28710.008,E2 -28710.008} C_VEL
LIN {X 0,Y 59.357,Z 440.937,A -85,B 0,C 180,E1 -28720.238,E2 -28720.238} C_VEL
LIN {X 0,Y 63.406,Z 434.806,A -85,B 0,C 180,E1 -28729.429,E2 -28729.429} C_VEL
LIN {X 0,Y 68.767,Z 427.144,A -85,B 0,C 180,E1 -28737.388,E2 -28737.388} C_VEL
LIN {X 0,Y 74.08,Z 419.271,A -85,B 0,C 180,E1 -28743.066,E2 -28743.066} C_VEL
LIN {X 0,Y 79.887,Z 409.693,A -85,B 0,C 180,E1 -28748.018,E2 -28748.018} C_VEL
LIN {X 0,Y 85.621,Z 399.033,A -85,B 0,C 180,E1 -28751.837,E2 -28751.837} C_VEL
LIN {X 0,Y 90.228,Z 388.654,A -85,B 0,C 180,E1 -28754.516,E2 -28754.516} C_VEL
LIN {X 0,Y 94.099,Z 377.457,A -85,B 0,C 180,E1 -28756.743,E2 -28756.743} C_VEL
LIN {X 0,Y 97.538,Z 365.182,A -85,B 0,C 180,E1 -28758.297,E2 -28758.297} C_VEL
LIN {X 0,Y 99.983,Z 352.076,A -85,B 0,C 180,E1 -28759.408,E2 -28759.408} C_VEL
LIN {X 0,Y 103.149,Z 320.862,A -85,B 0,C 180,E1 -28760.899,E2 -28760.899} C_VEL
LIN {X 0,Y 102.417,Z 318.822,A -85,B 0,C 180,E1 -28761.858,E2 -28761.858} C_VEL
LIN {X 0,Y 102.079,Z 318.975,A -85,B 0,C 180,E1 -28762.162,E2 -28762.162} C_VEL
LIN {X 0,Y 98.845,Z 326.221,A -85,B 0,C 180,E1 -28764.412,E2 -28764.412} C_VEL
LIN {X 0,Y 96.496,Z 330.423,A -85,B 0,C 180,E1 -28766.421,E2 -28766.421} C_VEL
LIN {X 0,Y 92.087,Z 346.496,A -85,B 0,C 180,E1 -28769.309,E2 -28769.309} C_VEL
LIN {X 0,Y 88.596,Z 356.671,A -85,B 0,C 180,E1 -28771.878,E2 -28771.878} C_VEL
LIN {X 0,Y 85.843,Z 362.852,A -85,B 0,C 180,E1 -28774.153,E2 -28774.153} C_VEL
LIN {X 0,Y 83.035,Z 367.752,A -85,B 0,C 180,E1 -28777.283,E2 -28777.283} C_VEL
LIN {X 0,Y 82.049,Z 369.309,A -85,B 0,C 180,E1 -28778.65,E2 -28778.65} C_VEL
LIN {X 0,Y 78.318,Z 377.196,A -85,B 0,C 180,E1 -28781.691,E2 -28781.691} C_VEL
LIN {X 0,Y 75.235,Z 382.888,A -85,B 0,C 180,E1 -28785.113,E2 -28785.113} C_VEL
LIN {X 0,Y 73.611,Z 385.774,A -85,B 0,C 180,E1 -28787.594,E2 -28787.594} C_VEL
LIN {X 0,Y 73.002,Z 386.855,A -85,B 0,C 180,E1 -28788.897,E2 -28788.897} C_VEL
LIN {X 0,Y 71.581,Z 389.599,A -85,B 0,C 180,E1 -28794.364,E2 -28794.364} C_VEL
LIN {X 0,Y 68.74,Z 396.426,A -85,B 0,C 180,E1 -28801.463,E2 -28801.463} C_VEL
LIN {X 0,Y 68.081,Z 399.286,A -85,B 0,C 180,E1 -28805.924,E2 -28805.924} C_VEL
LIN {X 0,Y 68.942,Z 401.257,A -85,B 0,C 180,E1 -28811.763,E2 -28811.763} C_VEL
LIN {X 0,Y 68.925,Z 404.39,A -85,B 0,C 180,E1 -28816.283,E2 -28816.283} C_VEL
LIN {X 0,Y 69.552,Z 409.683,A -85,B 0,C 180,E1 -28823.839,E2 -28823.839} C_VEL
LIN {X 0,Y 71.379,Z 412.944,A -85,B 0,C 180,E1 -28829.491,E2 -28829.491} C_VEL
LIN {X 0,Y 74.347,Z 415.28,A -85,B 0,C 180,E1 -28834.552,E2 -28834.552} C_VEL
LIN {X 0,Y 76.753,Z 415.695,A -85,B 0,C 180,E1 -28836.729,E2 -28836.729} C_VEL
LIN {X 0,Y 82.179,Z 422.846,A -85,B 0,C 180,E1 -28843.169,E2 -28843.169} C_VEL
LIN {X 0,Y 82.913,Z 423.712,A -85,B 0,C 180,E1 -28844.934,E2 -28844.934} C_VEL
LIN {X 0,Y 81.951,Z 422.833,A -85,B 0,C 180,E1 -28846.049,E2 -28846.049} C_VEL
LIN {X 0,Y 76.523,Z 428.143,A -85,B 0,C 180,E1 -28848.245,E2 -28848.245} C_VEL
LIN {X 0,Y 69.954,Z 435.102,A -85,B 0,C 180,E1 -28852.922,E2 -28852.922} C_VEL
LIN {X 0,Y 63.714,Z 442.055,A -85,B 0,C 180,E1 -28860.232,E2 -28860.232} C_VEL
LIN {X 0,Y 59.288,Z 447.634,A -85,B 0,C 180,E1 -28869.16,E2 -28869.16} C_VEL
LIN {X 0,Y 56.768,Z 452.024,A -85,B 0,C 180,E1 -28879.29,E2 -28879.29} C_VEL
LIN {X 0,Y 56.13,Z 455.326,A -85,B 0,C 180,E1 -28889.992,E2 -28889.992} C_VEL
LIN {X 0,Y 55.87,Z 456.892,A -85,B 0,C 180,E1 -28897.218,E2 -28897.218} C_VEL
LIN {X 0,Y 57.781,Z 458.84,A -85,B 0,C 180,E1 -28911.393,E2 -28911.393} C_VEL
LIN {X 0,Y 62.825,Z 459.169,A -85,B 0,C 180,E1 -28924.001,E2 -28924.001} C_VEL
LIN {X 0,Y 70.558,Z 457.996,A -85,B 0,C 180,E1 -28934.197,E2 -28934.197} C_VEL
LIN {X 0,Y 79.47,Z 455.406,A -85,B 0,C 180,E1 -28941.754,E2 -28941.754} C_VEL
LIN {X 0,Y 88.065,Z 452.008,A -85,B 0,C 180,E1 -28946.914,E2 -28946.914} C_VEL
LIN {X 0,Y 96.624,Z 447.787,A -85,B 0,C 180,E1 -28950.778,E2 -28950.778} C_VEL
LIN {X 0,Y 107.142,Z 441.402,A -85,B 0,C 180,E1 -28954.403,E2 -28954.403} C_VEL
LIN {X 0,Y 116.482,Z 434.435,A -85,B 0,C 180,E1 -28956.932,E2 -28956.932} C_VEL
LIN {X 0,Y 124.429,Z 427.361,A -85,B 0,C 180,E1 -28958.731,E2 -28958.731} C_VEL
LIN {X 0,Y 132.448,Z 418.819,A -85,B 0,C 180,E1 -28960.355,E2 -28960.355} C_VEL
LIN {X 0,Y 140.673,Z 408.304,A -85,B 0,C 180,E1 -28961.655,E2 -28961.655} C_VEL
LIN {X 0,Y 147.325,Z 397.857,A -85,B 0,C 180,E1 -28962.559,E2 -28962.559} C_VEL
LIN {X 0,Y 153.16,Z 386.23,A -85,B 0,C 180,E1 -28963.301,E2 -28963.301} C_VEL
LIN {X 0,Y 158.08,Z 373.272,A -85,B 0,C 180,E1 -28963.927,E2 -28963.927} C_VEL
LIN {X 0,Y 159.373,Z 368.878,A -85,B 0,C 180,E1 -28964.114,E2 -28964.114} C_VEL
LIN {X 0,Y 158.895,Z 366.694,A -85,B 0,C 180,E1 -28966.9,E2 -28966.9} C_VEL
LIN {X 0,Y 158.671,Z 365.144,A -85,B 0,C 180,E1 -28969.15,E2 -28969.15} C_VEL
LIN {X 0,Y 158.381,Z 364.476,A -85,B 0,C 180,E1 -28972.351,E2 -28972.351} C_VEL
LIN {X 0,Y 158.675,Z 364.724,A -85,B 0,C 180,E1 -28977.462,E2 -28977.462} C_VEL
LIN {X 0,Y 158.913,Z 367.635,A -85,B 0,C 180,E1 -28981.268,E2 -28981.268} C_VEL
LIN {X 0,Y 159.047,Z 368.894,A -85,B 0,C 180,E1 -28982.533,E2 -28982.533} C_VEL
LIN {X 0,Y 157.512,Z 373.829,A -85,B 0,C 180,E1 -28982.894,E2 -28982.894} C_VEL
LIN {X 0,Y 154.155,Z 382.563,A -85,B 0,C 180,E1 -28983.408,E2 -28983.408} C_VEL
LIN {X 0,Y 151.62,Z 387.981,A -85,B 0,C 180,E1 -28983.587,E2 -28983.587} C_VEL
LIN {X 0,Y 146.626,Z 396.526,A -85,B 0,C 180,E1 -28983.237,E2 -28983.237} C_VEL
LIN {X 0,Y 141.065,Z 404.628,A -85,B 0,C 180,E1 -28982.914,E2 -28982.914} C_VEL
LIN {X 0,Y 137.568,Z 409.301,A -85,B 0,C 180,E1 -28983.179,E2 -28983.179} C_VEL
LIN {X 0,Y 130.398,Z 417.911,A -85,B 0,C 180,E1 -28984.423,E2 -28984.423} C_VEL
LIN {X 0,Y 121.913,Z 426.345,A -85,B 0,C 180,E1 -28986.091,E2 -28986.091} C_VEL
LIN {X 0,Y 111.891,Z 434.529,A -85,B 0,C 180,E1 -28988.43,E2 -28988.43} C_VEL
LIN {X 0,Y 103.704,Z 440.031,A -85,B 0,C 180,E1 -28990.708,E2 -28990.708} C_VEL
LIN {X 0,Y 94.141,Z 445.344,A -85,B 0,C 180,E1 -28993.971,E2 -28993.971} C_VEL
LIN {X 0,Y 84.943,Z 449.392,A -85,B 0,C 180,E1 -28997.937,E2 -28997.937} C_VEL
LIN {X 0,Y 76.24,Z 452.311,A -85,B 0,C 180,E1 -29002.821,E2 -29002.821} C_VEL
LIN {X 0,Y 70.785,Z 453.658,A -85,B 0,C 180,E1 -29006.689,E2 -29006.689} C_VEL
LIN {X 0,Y 63.342,Z 454.887,A -85,B 0,C 180,E1 -29013.697,E2 -29013.697} C_VEL
LIN {X 0,Y 56.992,Z 455.152,A -85,B 0,C 180,E1 -29022.29,E2 -29022.29} C_VEL
LIN {X 0,Y 51.407,Z 454.182,A -85,B 0,C 180,E1 -29035.116,E2 -29035.116} C_VEL
LIN {X 0,Y 49.138,Z 452.809,A -85,B 0,C 180,E1 -29044.601,E2 -29044.601} C_VEL
LIN {X 0,Y 48.159,Z 450.183,A -85,B 0,C 180,E1 -29057.365,E2 -29057.365} C_VEL
LIN {X 0,Y 49.387,Z 446.511,A -85,B 0,C 180,E1 -29070.009,E2 -29070.009} C_VEL
LIN {X 0,Y 52.318,Z 441.728,A -85,B 0,C 180,E1 -29081.633,E2 -29081.633} C_VEL
LIN {X 0,Y 56.726,Z 435.703,A -85,B 0,C 180,E1 -29091.828,E2 -29091.828} C_VEL
LIN {X 0,Y 62.525,Z 428.201,A -85,B 0,C 180,E1 -29100.393,E2 -29100.393} C_VEL
LIN {X 0,Y 68.217,Z 420.503,A -85,B 0,C 180,E1 -29106.335,E2 -29106.335} C_VEL
LIN {X 0,Y 75.028,Z 410.105,A -85,B 0,C 180,E1 -29111.829,E2 -29111.829} C_VEL
LIN {X 0,Y 81.15,Z 399.401,A -85,B 0,C 180,E1 -29115.609,E2 -29115.609} C_VEL
LIN {X 0,Y 86.014,Z 389.036,A -85,B 0,C 180,E1 -29118.217,E2 -29118.217} C_VEL
LIN {X 0,Y 90.102,Z 377.848,A -85,B 0,C 180,E1 -29120.384,E2 -29120.384} C_VEL
LIN {X 0,Y 93.75,Z 365.38,A -85,B 0,C 180,E1 -29121.891,E2 -29121.891} C_VEL
LIN {X 0,Y 96.297,Z 352.27,A -85,B 0,C 180,E1 -29122.945,E2 -29122.945} C_VEL
LIN {X 0,Y 97.877,Z 338.106,A -85,B 0,C 180,E1 -29123.645,E2 -29123.645} C_VEL
LIN {X 0,Y 93.351,Z 352.555,A -85,B 0,C 180,E1 -29126.242,E2 -29126.242} C_VEL
LIN {X 0,Y 89,Z 362.697,A -85,B 0,C 180,E1 -29128.786,E2 -29128.786} C_VEL
LIN {X 0,Y 85.797,Z 368.429,A -85,B 0,C 180,E1 -29131.059,E2 -29131.059} C_VEL
LIN {X 0,Y 82.05,Z 373.803,A -85,B 0,C 180,E1 -29134.641,E2 -29134.641} C_VEL
LIN {X 0,Y 77.873,Z 381.294,A -85,B 0,C 180,E1 -29137.444,E2 -29137.444} C_VEL
LIN {X 0,Y 74.673,Z 386.28,A -85,B 0,C 180,E1 -29140.265,E2 -29140.265} C_VEL
LIN {X 0,Y 71.371,Z 391.04,A -85,B 0,C 180,E1 -29144.287,E2 -29144.287} C_VEL
LIN {X 0,Y 69.471,Z 393.621,A -85,B 0,C 180,E1 -29148.325,E2 -29148.325} C_VEL
LIN {X 0,Y 68.629,Z 394.92,A -85,B 0,C 180,E1 -29151.162,E2 -29151.162} C_VEL
LIN {X 0,Y 65.13,Z 401.356,A -85,B 0,C 180,E1 -29158.399,E2 -29158.399} C_VEL
LIN {X 0,Y 64.055,Z 404.161,A -85,B 0,C 180,E1 -29163.143,E2 -29163.143} C_VEL
LIN {X 0,Y 64.44,Z 407.007,A -85,B 0,C 180,E1 -29170.985,E2 -29170.985} C_VEL
LIN {X 0,Y 64.331,Z 414.185,A -85,B 0,C 180,E1 -29182.479,E2 -29182.479} C_VEL
LIN {X 0,Y 65.875,Z 417.352,A -85,B 0,C 180,E1 -29188.69,E2 -29188.69} C_VEL
LIN {X 0,Y 67.089,Z 418.65,A -85,B 0,C 180,E1 -29191.585,E2 -29191.585} C_VEL
LIN {X 0,Y 71.95,Z 421.262,A -85,B 0,C 180,E1 -29198.598,E2 -29198.598} C_VEL
LIN {X 0,Y 73.722,Z 423.249,A -85,B 0,C 180,E1 -29201.859,E2 -29201.859} C_VEL
LIN {X 0,Y 73.732,Z 424.872,A -85,B 0,C 180,E1 -29203.469,E2 -29203.469} C_VEL
LIN {X 0,Y 67.975,Z 430.65,A -85,B 0,C 180,E1 -29206.537,E2 -29206.537} C_VEL
LIN {X 0,Y 60.875,Z 437.904,A -85,B 0,C 180,E1 -29212.682,E2 -29212.682} C_VEL
LIN {X 0,Y 55.832,Z 443.276,A -85,B 0,C 180,E1 -29219.758,E2 -29219.758} C_VEL
LIN {X 0,Y 51.511,Z 448.547,A -85,B 0,C 180,E1 -29230.048,E2 -29230.048} C_VEL
LIN {X 0,Y 49.314,Z 452.652,A -85,B 0,C 180,E1 -29241.797,E2 -29241.797} C_VEL
LIN {X 0,Y 49.035,Z 454.808,A -85,B 0,C 180,E1 -29249.991,E2 -29249.991} C_VEL
LIN {X 0,Y 48.83,Z 456.414,A -85,B 0,C 180,E1 -29258.266,E2 -29258.266} C_VEL
LIN {X 0,Y 51.223,Z 458.438,A -85,B 0,C 180,E1 -29274.297,E2 -29274.297} C_VEL
LIN {X 0,Y 53.716,Z 458.86,A -85,B 0,C 180,E1 -29281.547,E2 -29281.547} C_VEL
LIN {X 0,Y 61.109,Z 458.512,A -85,B 0,C 180,E1 -29293.624,E2 -29293.624} C_VEL
LIN {X 0,Y 70.626,Z 456.653,A -85,B 0,C 180,E1 -29302.747,E2 -29302.747} C_VEL
LIN {X 0,Y 75.908,Z 455.09,A -85,B 0,C 180,E1 -29306.425,E2 -29306.425} C_VEL
LIN {X 0,Y 84.387,Z 451.988,A -85,B 0,C 180,E1 -29310.971,E2 -29310.971} C_VEL
LIN {X 0,Y 93.369,Z 447.856,A -85,B 0,C 180,E1 -29314.578,E2 -29314.578} C_VEL
LIN {X 0,Y 104.275,Z 441.568,A -85,B 0,C 180,E1 -29317.919,E2 -29317.919} C_VEL
LIN {X 0,Y 113.89,Z 434.744,A -85,B 0,C 180,E1 -29320.217,E2 -29320.217} C_VEL
LIN {X 0,Y 122.036,Z 427.796,A -85,B 0,C 180,E1 -29321.835,E2 -29321.835} C_VEL
LIN {X 0,Y 130.244,Z 419.43,A -85,B 0,C 180,E1 -29323.282,E2 -29323.282} C_VEL
LIN {X 0,Y 138.611,Z 409.102,A -85,B 0,C 180,E1 -29324.429,E2 -29324.429} C_VEL
LIN {X 0,Y 146.212,Z 397.497,A -85,B 0,C 180,E1 -29325.306,E2 -29325.306} C_VEL
LIN {X 0,Y 152.131,Z 385.861,A -85,B 0,C 180,E1 -29325.949,E2 -29325.949} C_VEL
LIN {X 0,Y 156.601,Z 374.431,A -85,B 0,C 180,E1 -29326.433,E2 -29326.433} C_VEL
LIN {X 0,Y 156.742,Z 373.752,A -85,B 0,C 180,E1 -29326.716,E2 -29326.716} C_VEL
LIN {X 0,Y 156.591,Z 371.849,A -85,B 0,C 180,E1 -29329.658,E2 -29329.658} C_VEL
